LIN {X -0.027,Y -194.298,Z 687.966,A 0.000,B 0.000,C 90.000,E1 353.799} C_DIS
LIN {X 0.100,Y -197.858,Z 687.934,A 0.000,B 0.000,C 90.000,E1 348.049} C_DIS
LIN {X -0.011,Y -201.599,Z 687.911,A 0.000,B 0.000,C 90.000,E1 344.031} C_DIS
LIN {X 0.020,Y -206.301,Z 687.889,A 0.000,B 0.000,C 90.000,E1 340.007} C_DIS
LIN {X -0.035,Y -211.829,Z 687.867,A 0.000,B 0.000,C 90.000,E1 336.049} C_DIS
LIN {X 0.046,Y -218.045,Z 687.845,A 0.000,B 0.000,C 90.000,E1 332.103} C_DIS
LIN {X -0.027,Y -225.043,Z 687.824,A 0.000,B 0.000,C 90.000,E1 328.250} C_DIS
LIN {X 0.020,Y -231.035,Z 687.807,A 0.000,B 0.000,C 90.000,E1 325.182} C_DIS
LIN {X 0.033,Y -239.102,Z 687.786,A 0.000,B 0.000,C 90.000,E1 321.412} C_DIS
LIN {X 0.002,Y -248.003,Z 687.765,A 0.000,B 0.000,C 90.000,E1 317.715} C_DIS
LIN {X 0.037,Y -256.957,Z 687.747,A 0.000,B 0.000,C 90.000,E1 314.433} C_DIS
LIN {X 0.065,Y -267.947,Z 687.727,A 0.000,B 0.000,C 90.000,E1 310.862} C_DIS
LIN {X 0.020,Y -279.022,Z 687.710,A 0.000,B 0.000,C 90.000,E1 307.729} C_DIS
LIN {X -0.029,Y -292.675,Z 687.691,A 0.000,B 0.000,C 90.000,E1 304.326} C_DIS
LIN {X -0.050,Y -307.715,Z 687.672,A 0.000,B 0.000,C 90.000,E1 301.003} C_DIS
LIN {X -0.132,Y -319.136,Z 687.660,A 0.000,B 0.000,C 90.000,E1 298.743} C_DIS
LIN {X 0.084,Y -334.892,Z 687.644,A 0.000,B 0.000,C 90.000,E1 295.848} C_DIS
LIN {X 0.026,Y -351.489,Z 687.628,A 0.000,B 0.000,C 90.000,E1 293.078} C_DIS
LIN {X 0.026,Y -369.148,Z 687.613,A 0.000,B 0.000,C 90.000,E1 290.375} C_DIS
LIN {X 0.146,Y -381.918,Z 687.603,A 0.000,B 0.000,C 90.000,E1 288.598} C_DIS
LIN {X 0.106,Y -400.402,Z 687.591,A 0.000,B 0.000,C 90.000,E1 286.315} C_DIS
LIN {X -0.150,Y -412.016,Z 687.583,A 0.000,B 0.000,C 90.000,E1 284.954} C_DIS
LIN {X 0.167,Y -423.397,Z 687.575,A 0.000,B 0.000,C 90.000,E1 283.536} C_DIS
LIN {X 0.161,Y -434.292,Z 687.568,A 0.000,B 0.000,C 90.000,E1 282.187} C_DIS
LIN {X 0.099,Y -442.576,Z 687.562,A 0.000,B 0.000,C 90.000,E1 281.130} C_DIS
LIN {X -0.097,Y -460.504,Z 687.549,A 0.000,B 0.000,C 90.000,E1 278.803} C_DIS
LIN {X -0.165,Y -470.432,Z 687.542,A 0.000,B 0.000,C 90.000,E1 277.530} C_DIS
LIN {X -0.225,Y -475.757,Z 687.537,A 0.000,B 0.000,C 90.000,E1 276.777} C_DIS
LIN {X 0.239,Y -480.127,Z 687.533,A 0.000,B 0.000,C 90.000,E1 275.967} C_DIS
LIN {X 0.212,Y -483.506,Z 687.529,A 0.000,B 0.000,C 90.000,E1 275.220} C_DIS
LIN {X -0.094,Y -485.203,Z 687.526,A 0.000,B 0.000,C 90.000,E1 274.759} C_DIS
LIN {X 0.050,Y -486.474,Z 687.524,A 0.000,B 0.000,C 90.000,E1 274.245} C_DIS
LIN {X 0.241,Y -487.342,Z 687.521,A 0.000,B 0.000,C 90.000,E1 273.726} C_DIS
LIN {X -0.077,Y -487.894,Z 687.518,A 0.000,B 0.000,C 90.000,E1 273.269} C_DIS
LIN {X 0.122,Y -488.076,Z 687.515,A 0.000,B 0.000,C 90.000,E1 272.751} C_DIS
LIN {X -0.186,Y -487.966,Z 687.513,A 0.000,B 0.000,C 90.000,E1 272.293} C_DIS
LIN {X 0.013,Y -487.497,Z 687.510,A 0.000,B 0.000,C 90.000,E1 271.776} C_DIS
LIN {X 0.193,Y -486.720,Z 687.507,A 0.000,B 0.000,C 90.000,E1 271.260} C_DIS
LIN {X -0.115,Y -485.520,Z 687.504,A 0.000,B 0.000,C 90.000,E1 270.802} C_DIS
LIN {X 0.061,Y -483.850,Z 687.502,A 0.000,B 0.000,C 90.000,E1 270.286} C_DIS
LIN {X 0.228,Y -481.575,Z 687.499,A 0.000,B 0.000,C 90.000,E1 269.771} C_DIS
LIN {X 0.063,Y -480.227,Z 687.497,A 0.000,B 0.000,C 90.000,E1 269.542} C_DIS
LIN {X 0.206,Y -476.929,Z 687.495,A 0.000,B 0.000,C 90.000,E1 269.026} C_DIS
LIN {X -0.145,Y -472.762,Z 687.492,A 0.000,B 0.000,C 90.000,E1 268.568} C_DIS
LIN {X 0.005,Y -467.541,Z 687.489,A 0.000,B 0.000,C 90.000,E1 268.051} C_DIS
LIN {X -0.015,Y -461.447,Z 687.487,A 0.000,B 0.000,C 90.000,E1 267.593} C_DIS
LIN {X 0.115,Y -458.008,Z 687.485,A 0.000,B 0.000,C 90.000,E1 267.364} C_DIS
LIN {X 0.027,Y -451.055,Z 687.483,A 0.000,B 0.000,C 90.000,E1 267.020} C_DIS
LIN {X 0.028,Y -443.900,Z 687.482,A 0.000,B 0.000,C 90.000,E1 266.731} C_DIS
LIN {X 0.017,Y -436.381,Z 687.481,A 0.000,B 0.000,C 90.000,E1 266.502} C_DIS
LIN {X 0.206,Y -432.252,Z 687.480,A 0.000,B 0.000,C 90.000,E1 266.388} C_DIS
LIN {X 0.052,Y -421.992,Z 687.479,A 0.000,B 0.000,C 90.000,E1 266.274} C_DIS
LIN {X -0.200,Y -415.695,Z 687.479,A 0.000,B 0.000,C 90.000,E1 266.274} C_DIS
LIN {X 0.071,Y -180.932,Z 687.479,A 0.000,B 0.000,C 90.000,E1 266.216} C_DIS
LIN {X -0.053,Y -180.770,Z 687.471,A 0.000,B 0.000,C 90.000,E1 264.723} C_DIS
LIN {X -0.015,Y -178.987,Z 687.444,A 0.000,B 0.000,C 90.000,E1 259.982} C_DIS
LIN {X -0.004,Y -177.967,Z 687.435,A 0.000,B 0.000,C 90.000,E1 258.285} C_DIS
LIN {X 0.015,Y -175.610,Z 687.411,A 0.000,B 0.000,C 90.000,E1 254.031} C_DIS
LIN {X 0.027,Y -172.332,Z 687.388,A 0.000,B 0.000,C 90.000,E1 249.752} C_DIS
LIN {X 0.006,Y -171.808,Z 687.383,A 0.000,B 0.000,C 90.000,E1 248.901} C_DIS
LIN {X 0.013,Y -170.270,Z 687.373,A 0.000,B 0.000,C 90.000,E1 247.177} C_DIS
LIN {X -0.051,Y -166.812,Z 687.349,A 0.000,B 0.000,C 90.000,E1 242.871} C_DIS
LIN {X 0.007,Y -162.794,Z 687.325,A 0.000,B 0.000,C 90.000,E1 238.486} C_DIS
LIN {X 0.067,Y -161.481,Z 687.315,A 0.000,B 0.000,C 90.000,E1 236.707} C_DIS
LIN {X -0.017,Y -157.477,Z 687.291,A 0.000,B 0.000,C 90.000,E1 232.316} C_DIS
LIN {X 0.040,Y -155.493,Z 687.276,A 0.000,B 0.000,C 90.000,E1 229.622} C_DIS
LIN {X -0.028,Y -151.799,Z 687.251,A 0.000,B 0.000,C 90.000,E1 225.162} C_DIS
LIN {X -0.015,Y -150.008,Z 687.236,A 0.000,B 0.000,C 90.000,E1 222.447} C_DIS
LIN {X 0.017,Y -146.834,Z 687.211,A 0.000,B 0.000,C 90.000,E1 217.890} C_DIS
LIN {X 0.003,Y -145.416,Z 687.195,A 0.000,B 0.000,C 90.000,E1 215.152} C_DIS
LIN {X 0.038,Y -142.844,Z 687.170,A 0.000,B 0.000,C 90.000,E1 210.541} C_DIS
LIN {X -0.032,Y -141.458,Z 687.149,A 0.000,B 0.000,C 90.000,E1 206.873} C_DIS
LIN {X 0.008,Y -139.374,Z 687.113,A 0.000,B 0.000,C 90.000,E1 200.355} C_DIS
LIN {X -0.051,Y -138.825,Z 687.098,A 0.000,B 0.000,C 90.000,E1 197.583} C_DIS
LIN {X 0.038,Y -138.353,Z 687.056,A 0.000,B 0.000,C 90.000,E1 190.074} C_DIS
LIN {X 0.012,Y -139.531,Z 687.004,A 0.000,B 0.000,C 90.000,E1 180.745} C_DIS
LIN {X -0.036,Y -141.212,Z 686.973,A 0.000,B 0.000,C 90.000,E1 175.179} C_DIS
LIN {X 0.065,Y -142.585,Z 686.958,A 0.000,B 0.000,C 90.000,E1 172.356} C_DIS
LIN {X 0.019,Y -144.883,Z 686.932,A 0.000,B 0.000,C 90.000,E1 167.757} C_DIS
LIN {X -0.028,Y -147.510,Z 686.912,A 0.000,B 0.000,C 90.000,E1 164.102} C_DIS
LIN {X 0.047,Y -150.103,Z 686.891,A 0.000,B 0.000,C 90.000,E1 160.423} C_DIS
LIN {X 0.059,Y -153.461,Z 686.871,A 0.000,B 0.000,C 90.000,E1 156.794} C_DIS
LIN {X -0.089,Y -157.823,Z 686.846,A 0.000,B 0.000,C 90.000,E1 152.359} C_DIS
LIN {X -0.057,Y -162.107,Z 686.826,A 0.000,B 0.000,C 90.000,E1 148.791} C_DIS
LIN {X -0.033,Y -166.308,Z 686.807,A 0.000,B 0.000,C 90.000,E1 145.261} C_DIS
LIN {X 0.069,Y -171.325,Z 686.788,A 0.000,B 0.000,C 90.000,E1 141.743} C_DIS
LIN {X -0.003,Y -176.225,Z 686.768,A 0.000,B 0.000,C 90.000,E1 138.324} C_DIS
LIN {X -0.009,Y -180.504,Z 686.754,A 0.000,B 0.000,C 90.000,E1 135.769} C_DIS
LIN {X 0.097,Y -185.907,Z 686.736,A 0.000,B 0.000,C 90.000,E1 132.366} C_DIS
LIN {X 0.078,Y -191.207,Z 686.719,A 0.000,B 0.000,C 90.000,E1 129.483} C_DIS
LIN {X 0.075,Y -289.233,Z 686.719,A 0.000,B 0.000,C 90.000,E1 129.483} C_DIS
LIN {X 0.007,Y -295.104,Z 686.718,A 0.000,B 0.000,C 90.000,E1 129.277} C_DIS
LIN {X -0.016,Y -297.647,Z 686.717,A 0.000,B 0.000,C 90.000,E1 129.072} C_DIS
LIN {X -0.033,Y -301.459,Z 686.714,A 0.000,B 0.000,C 90.000,E1 128.588} C_DIS
LIN {X -0.038,Y -303.267,Z 686.713,A 0.000,B 0.000,C 90.000,E1 128.257} C_DIS
LIN {X -0.094,Y -304.679,Z 686.711,A 0.000,B 0.000,C 90.000,E1 127.935} C_DIS
LIN {X 0.123,Y -306.687,Z 686.707,A 0.000,B 0.000,C 90.000,E1 127.237} C_DIS
LIN {X 0.057,Y -316.400,Z 686.689,A 0.000,B 0.000,C 90.000,E1 123.992} C_DIS
LIN {X -0.038,Y -326.433,Z 686.673,A 0.000,B 0.000,C 90.000,E1 121.131} C_DIS
LIN {X 0.089,Y -337.794,Z 686.657,A 0.000,B 0.000,C 90.000,E1 118.281} C_DIS
LIN {X -0.088,Y -350.581,Z 686.642,A 0.000,B 0.000,C 90.000,E1 115.540} C_DIS
LIN {X -0.118,Y -363.240,Z 686.628,A 0.000,B 0.000,C 90.000,E1 113.131} C_DIS
LIN {X 0.082,Y -377.206,Z 686.615,A 0.000,B 0.000,C 90.000,E1 110.737} C_DIS
LIN {X 0.160,Y -392.584,Z 686.602,A 0.000,B 0.000,C 90.000,E1 108.417} C_DIS
LIN {X -0.133,Y -409.482,Z 686.590,A 0.000,B 0.000,C 90.000,E1 106.205} C_DIS
LIN {X -0.128,Y -428.026,Z 686.578,A 0.000,B 0.000,C 90.000,E1 104.008} C_DIS
LIN {X 0.121,Y -447.934,Z 686.566,A 0.000,B 0.000,C 90.000,E1 101.883} C_DIS
LIN {X 0.120,Y -468.437,Z 686.555,A 0.000,B 0.000,C 90.000,E1 99.962} C_DIS
LIN {X 0.167,Y -470.660,Z 686.554,A 0.000,B 0.000,C 90.000,E1 99.726} C_DIS
LIN {X -0.052,Y -472.481,Z 686.553,A 0.000,B 0.000,C 90.000,E1 99.500} C_DIS
LIN {X -0.192,Y -473.850,Z 686.551,A 0.000,B 0.000,C 90.000,E1 99.265} C_DIS
LIN {X -0.079,Y -475.584,Z 686.549,A 0.000,B 0.000,C 90.000,E1 98.746} C_DIS
LIN {X 0.115,Y -476.240,Z 686.546,A 0.000,B 0.000,C 90.000,E1 98.219} C_DIS
LIN {X -0.224,Y -475.928,Z 686.543,A 0.000,B 0.000,C 90.000,E1 97.757} C_DIS
LIN {X -0.085,Y -474.605,Z 686.540,A 0.000,B 0.000,C 90.000,E1 97.239} C_DIS
LIN {X 0.247,Y -473.499,Z 686.539,A 0.000,B 0.000,C 90.000,E1 96.947} C_DIS
LIN {X 0.053,Y -472.021,Z 686.537,A 0.000,B 0.000,C 90.000,E1 96.720} C_DIS
LIN {X 0.219,Y -453.746,Z 686.522,A 0.000,B 0.000,C 90.000,E1 93.898} C_DIS
LIN {X 0.187,Y -437.541,Z 686.506,A 0.000,B 0.000,C 90.000,E1 91.031} C_DIS
LIN {X 0.114,Y -430.195,Z 686.498,A 0.000,B 0.000,C 90.000,E1 89.714} C_DIS
LIN {X 0.071,Y -420.954,Z 686.490,A 0.000,B 0.000,C 90.000,E1 88.108} C_DIS
LIN {X 0.059,Y -408.465,Z 686.477,A 0.000,B 0.000,C 90.000,E1 85.927} C_DIS
LIN {X 0.177,Y -395.953,Z 686.465,A 0.000,B 0.000,C 90.000,E1 83.685} C_DIS
LIN {X 0.115,Y -382.283,Z 686.451,A 0.000,B 0.000,C 90.000,E1 81.141} C_DIS
LIN {X 0.186,Y -370.570,Z 686.438,A 0.000,B 0.000,C 90.000,E1 78.814} C_DIS
LIN {X 0.043,Y -356.463,Z 686.422,A 0.000,B 0.000,C 90.000,E1 75.880} C_DIS
LIN {X -0.177,Y -345.659,Z 686.408,A 0.000,B 0.000,C 90.000,E1 73.504} C_DIS
LIN {X -0.138,Y -333.972,Z 686.393,A 0.000,B 0.000,C 90.000,E1 70.732} C_DIS
LIN {X 0.076,Y -319.540,Z 686.372,A 0.000,B 0.000,C 90.000,E1 66.922} C_DIS
LIN {X 0.089,Y -307.949,Z 686.352,A 0.000,B 0.000,C 90.000,E1 63.384} C_DIS
LIN {X -0.001,Y -298.482,Z 686.334,A 0.000,B 0.000,C 90.000,E1 60.127} C_DIS
LIN {X 0.061,Y -289.725,Z 686.316,A 0.000,B 0.000,C 90.000,E1 56.786} C_DIS
LIN {X -0.091,Y -283.065,Z 686.301,A 0.000,B 0.000,C 90.000,E1 54.116} C_DIS
LIN {X -0.074,Y -278.087,Z 686.289,A 0.000,B 0.000,C 90.000,E1 52.065} C_DIS
LIN {X -0.031,Y -272.884,Z 686.278,A 0.000,B 0.000,C 90.000,E1 49.989} C_DIS
LIN {X -0.112,Y -267.376,Z 686.266,A 0.000,B 0.000,C 90.000,E1 47.919} C_DIS
LIN {X -0.112,Y -261.484,Z 686.254,A 0.000,B 0.000,C 90.000,E1 45.810} C_DIS
LIN {X 0.132,Y -255.455,Z 686.242,A 0.000,B 0.000,C 90.000,E1 43.623} C_DIS
LIN {X -0.093,Y -249.280,Z 686.231,A 0.000,B 0.000,C 90.000,E1 41.515} C_DIS
LIN {X 0.129,Y -242.951,Z 686.218,A 0.000,B 0.000,C 90.000,E1 39.277} C_DIS
LIN {X 0.026,Y -232.833,Z 686.198,A 0.000,B 0.000,C 90.000,E1 35.598} C_DIS
LIN {X -0.033,Y -225.322,Z 686.181,A 0.000,B 0.000,C 90.000,E1 32.594} C_DIS
LIN {X -0.067,Y -218.723,Z 686.164,A 0.000,B 0.000,C 90.000,E1 29.539} C_DIS
LIN {X 0.010,Y -212.830,Z 686.147,A 0.000,B 0.000,C 90.000,E1 26.411} C_DIS
LIN {X 0.035,Y -207.796,Z 686.129,A 0.000,B 0.000,C 90.000,E1 23.259} C_DIS
LIN {X 0.076,Y -202.633,Z 686.107,A 0.000,B 0.000,C 90.000,E1 19.268} C_DIS
LIN {X 0.080,Y -198.620,Z 686.085,A 0.000,B 0.000,C 90.000,E1 15.245} C_DIS
LIN {X 0.109,Y -195.196,Z 686.058,A 0.000,B 0.000,C 90.000,E1 10.366} C_DIS
LIN {X -0.002,Y -192.827,Z 686.017,A 0.000,B 0.000,C 90.000,E1 3.037} C_DIS
LIN {X -0.022,Y -194.394,Z 685.966,A 0.000,B 0.000,C 90.000,E1 353.799} C_DIS
LIN {X 0.109,Y -197.929,Z 685.934,A 0.000,B 0.000,C 90.000,E1 348.049} C_DIS
LIN {X 0.001,Y -201.671,Z 685.911,A 0.000,B 0.000,C 90.000,E1 344.031} C_DIS
LIN {X 0.034,Y -206.368,Z 685.889,A 0.000,B 0.000,C 90.000,E1 340.007} C_DIS
LIN {X -0.019,Y -211.878,Z 685.867,A 0.000,B 0.000,C 90.000,E1 336.049} C_DIS
LIN {X 0.064,Y -218.099,Z 685.845,A 0.000,B 0.000,C 90.000,E1 332.103} C_DIS
LIN {X -0.007,Y -225.100,Z 685.824,A 0.000,B 0.000,C 90.000,E1 328.250} C_DIS
LIN {X 0.042,Y -231.081,Z 685.807,A 0.000,B 0.000,C 90.000,E1 325.182} C_DIS
LIN {X 0.057,Y -239.126,Z 685.786,A 0.000,B 0.000,C 90.000,E1 321.412} C_DIS
LIN {X 0.029,Y -248.003,Z 685.765,A 0.000,B 0.000,C 90.000,E1 317.715} C_DIS
LIN {X -0.096,Y -258.017,Z 685.745,A 0.000,B 0.000,C 90.000,E1 314.109} C_DIS
LIN {X -0.044,Y -269.115,Z 685.725,A 0.000,B 0.000,C 90.000,E1 310.539} C_DIS
LIN {X -0.013,Y -280.316,Z 685.708,A 0.000,B 0.000,C 90.000,E1 307.397} C_DIS
LIN {X -0.011,Y -294.084,Z 685.689,A 0.000,B 0.000,C 90.000,E1 303.992} C_DIS
LIN {X 0.019,Y -309.250,Z 685.670,A 0.000,B 0.000,C 90.000,E1 300.669} C_DIS
LIN {X -0.091,Y -326.003,Z 685.652,A 0.000,B 0.000,C 90.000,E1 297.462} C_DIS
LIN {X -0.121,Y -342.118,Z 685.637,A 0.000,B 0.000,C 90.000,E1 294.643} C_DIS
LIN {X -0.018,Y -363.058,Z 685.618,A 0.000,B 0.000,C 90.000,E1 291.280} C_DIS
LIN {X -0.018,Y -375.260,Z 685.608,A 0.000,B 0.000,C 90.000,E1 289.504} C_DIS
LIN {X -0.083,Y -395.523,Z 685.594,A 0.000,B 0.000,C 90.000,E1 286.913} C_DIS
LIN {X 0.174,Y -409.571,Z 685.585,A 0.000,B 0.000,C 90.000,E1 285.190} C_DIS
LIN {X -0.216,Y -423.240,Z 685.575,A 0.000,B 0.000,C 90.000,E1 283.592} C_DIS
LIN {X -0.237,Y -434.130,Z 685.568,A 0.000,B 0.000,C 90.000,E1 282.243} C_DIS
LIN {X 0.123,Y -442.396,Z 685.562,A 0.000,B 0.000,C 90.000,E1 281.130} C_DIS
LIN {X 0.202,Y -462.319,Z 685.547,A 0.000,B 0.000,C 90.000,E1 278.511} C_DIS
LIN {X -0.147,Y -470.230,Z 685.542,A 0.000,B 0.000,C 90.000,E1 277.530} C_DIS
LIN {X -0.208,Y -475.560,Z 685.538,A 0.000,B 0.000,C 90.000,E1 276.777} C_DIS
LIN {X -0.082,Y -478.576,Z 685.535,A 0.000,B 0.000,C 90.000,E1 276.258} C_DIS
LIN {X -0.119,Y -482.284,Z 685.531,A 0.000,B 0.000,C 90.000,E1 275.511} C_DIS
LIN {X -0.082,Y -484.984,Z 685.526,A 0.000,B 0.000,C 90.000,E1 274.759} C_DIS
LIN {X 0.060,Y -486.297,Z 685.524,A 0.000,B 0.000,C 90.000,E1 274.245} C_DIS
LIN {X -0.235,Y -487.161,Z 685.521,A 0.000,B 0.000,C 90.000,E1 273.784} C_DIS
LIN {X -0.070,Y -487.709,Z 685.518,A 0.000,B 0.000,C 90.000,E1 273.269} C_DIS
LIN {X 0.129,Y -487.921,Z 685.515,A 0.000,B 0.000,C 90.000,E1 272.751} C_DIS
LIN {X -0.180,Y -487.837,Z 685.513,A 0.000,B 0.000,C 90.000,E1 272.293} C_DIS
LIN {X 0.018,Y -487.439,Z 685.510,A 0.000,B 0.000,C 90.000,E1 271.776} C_DIS
LIN {X 0.198,Y -486.637,Z 685.507,A 0.000,B 0.000,C 90.000,E1 271.260} C_DIS
LIN {X -0.110,Y -485.469,Z 685.504,A 0.000,B 0.000,C 90.000,E1 270.802} C_DIS
LIN {X 0.065,Y -483.831,Z 685.502,A 0.000,B 0.000,C 90.000,E1 270.286} C_DIS
LIN {X 0.231,Y -481.597,Z 685.499,A 0.000,B 0.000,C 90.000,E1 269.771} C_DIS
LIN {X -0.097,Y -478.673,Z 685.496,A 0.000,B 0.000,C 90.000,E1 269.312} C_DIS
LIN {X 0.208,Y -476.971,Z 685.495,A 0.000,B 0.000,C 90.000,E1 269.026} C_DIS
LIN {X -0.142,Y -472.795,Z 685.492,A 0.000,B 0.000,C 90.000,E1 268.568} C_DIS
LIN {X 0.013,Y -467.555,Z 685.489,A 0.000,B 0.000,C 90.000,E1 268.051} C_DIS
LIN {X -0.015,Y -461.461,Z 685.487,A 0.000,B 0.000,C 90.000,E1 267.593} C_DIS
LIN {X 0.051,Y -454.772,Z 685.484,A 0.000,B 0.000,C 90.000,E1 267.192} C_DIS
LIN {X -0.226,Y -447.733,Z 685.483,A 0.000,B 0.000,C 90.000,E1 266.906} C_DIS
LIN {X 0.004,Y -440.474,Z 685.481,A 0.000,B 0.000,C 90.000,E1 266.617} C_DIS
LIN {X 0.194,Y -432.352,Z 685.480,A 0.000,B 0.000,C 90.000,E1 266.388} C_DIS
LIN {X 0.061,Y -422.993,Z 685.479,A 0.000,B 0.000,C 90.000,E1 266.274} C_DIS
LIN {X 0.153,Y -415.264,Z 685.479,A 0.000,B 0.000,C 90.000,E1 266.216} C_DIS
LIN {X 0.043,Y -180.931,Z 685.479,A 0.000,B 0.000,C 90.000,E1 266.216} C_DIS
LIN {X -0.061,Y -180.769,Z 685.471,A 0.000,B 0.000,C 90.000,E1 264.723} C_DIS
LIN {X -0.024,Y -178.986,Z 685.444,A 0.000,B 0.000,C 90.000,E1 259.982} C_DIS
LIN {X -0.012,Y -177.965,Z 685.435,A 0.000,B 0.000,C 90.000,E1 258.285} C_DIS
LIN {X 0.007,Y -175.608,Z 685.411,A 0.000,B 0.000,C 90.000,E1 254.031} C_DIS
LIN {X 0.020,Y -172.330,Z 685.388,A 0.000,B 0.000,C 90.000,E1 249.752} C_DIS
LIN {X -0.001,Y -171.807,Z 685.383,A 0.000,B 0.000,C 90.000,E1 248.901} C_DIS
LIN {X 0.006,Y -170.268,Z 685.373,A 0.000,B 0.000,C 90.000,E1 247.177} C_DIS
LIN {X -0.058,Y -166.810,Z 685.349,A 0.000,B 0.000,C 90.000,E1 242.871} C_DIS
LIN {X 0.000,Y -162.792,Z 685.325,A 0.000,B 0.000,C 90.000,E1 238.486} C_DIS
LIN {X 0.060,Y -161.480,Z 685.315,A 0.000,B 0.000,C 90.000,E1 236.707} C_DIS
LIN {X -0.024,Y -157.475,Z 685.291,A 0.000,B 0.000,C 90.000,E1 232.316} C_DIS
LIN {X 0.033,Y -155.490,Z 685.276,A 0.000,B 0.000,C 90.000,E1 229.622} C_DIS
LIN {X -0.034,Y -151.797,Z 685.251,A 0.000,B 0.000,C 90.000,E1 225.162} C_DIS
LIN {X -0.021,Y -150.006,Z 685.236,A 0.000,B 0.000,C 90.000,E1 222.447} C_DIS
LIN {X 0.010,Y -146.833,Z 685.211,A 0.000,B 0.000,C 90.000,E1 217.890} C_DIS
LIN {X -0.004,Y -145.413,Z 685.195,A 0.000,B 0.000,C 90.000,E1 215.152} C_DIS
LIN {X 0.032,Y -142.843,Z 685.170,A 0.000,B 0.000,C 90.000,E1 210.541} C_DIS
LIN {X -0.039,Y -141.457,Z 685.149,A 0.000,B 0.000,C 90.000,E1 206.873} C_DIS
LIN {X 0.001,Y -139.373,Z 685.113,A 0.000,B 0.000,C 90.000,E1 200.355} C_DIS
LIN {X -0.057,Y -138.824,Z 685.098,A 0.000,B 0.000,C 90.000,E1 197.583} C_DIS
LIN {X 0.032,Y -138.353,Z 685.056,A 0.000,B 0.000,C 90.000,E1 190.074} C_DIS
LIN {X 0.005,Y -139.532,Z 685.004,A 0.000,B 0.000,C 90.000,E1 180.745} C_DIS
LIN {X -0.042,Y -141.212,Z 684.973,A 0.000,B 0.000,C 90.000,E1 175.179} C_DIS
LIN {X 0.058,Y -142.586,Z 684.958,A 0.000,B 0.000,C 90.000,E1 172.356} C_DIS
LIN {X 0.012,Y -144.885,Z 684.932,A 0.000,B 0.000,C 90.000,E1 167.757} C_DIS
LIN {X -0.035,Y -147.512,Z 684.912,A 0.000,B 0.000,C 90.000,E1 164.102} C_DIS
LIN {X 0.040,Y -150.106,Z 684.891,A 0.000,B 0.000,C 90.000,E1 160.423} C_DIS
LIN {X 0.053,Y -153.462,Z 684.871,A 0.000,B 0.000,C 90.000,E1 156.794} C_DIS
LIN {X -0.096,Y -157.826,Z 684.846,A 0.000,B 0.000,C 90.000,E1 152.359} C_DIS
LIN {X 0.074,Y -162.110,Z 684.826,A 0.000,B 0.000,C 90.000,E1 148.742} C_DIS
LIN {X -0.040,Y -166.311,Z 684.807,A 0.000,B 0.000,C 90.000,E1 145.261} C_DIS
LIN {X 0.061,Y -171.329,Z 684.788,A 0.000,B 0.000,C 90.000,E1 141.743} C_DIS
LIN {X -0.010,Y -176.229,Z 684.768,A 0.000,B 0.000,C 90.000,E1 138.324} C_DIS
LIN {X 0.109,Y -180.509,Z 684.754,A 0.000,B 0.000,C 90.000,E1 135.729} C_DIS
LIN {X 0.089,Y -185.911,Z 684.736,A 0.000,B 0.000,C 90.000,E1 132.366} C_DIS
LIN {X 0.006,Y -191.183,Z 684.720,A 0.000,B 0.000,C 90.000,E1 129.519} C_DIS
LIN {X -0.034,Y -288.963,Z 684.720,A 0.000,B 0.000,C 90.000,E1 129.519} C_DIS
LIN {X 0.020,Y -290.728,Z 684.719,A 0.000,B 0.000,C 90.000,E1 129.483} C_DIS
LIN {X -0.005,Y -295.281,Z 684.718,A 0.000,B 0.000,C 90.000,E1 129.277} C_DIS
LIN {X -0.028,Y -297.754,Z 684.717,A 0.000,B 0.000,C 90.000,E1 129.072} C_DIS
LIN {X 0.129,Y -301.574,Z 684.714,A 0.000,B 0.000,C 90.000,E1 128.543} C_DIS
LIN {X -0.112,Y -303.342,Z 684.712,A 0.000,B 0.000,C 90.000,E1 128.257} C_DIS
LIN {X 0.073,Y -304.726,Z 684.711,A 0.000,B 0.000,C 90.000,E1 127.890} C_DIS
LIN {X 0.034,Y -308.532,Z 684.703,A 0.000,B 0.000,C 90.000,E1 126.583} C_DIS
LIN {X -0.153,Y -318.544,Z 684.685,A 0.000,B 0.000,C 90.000,E1 123.372} C_DIS
LIN {X 0.086,Y -328.870,Z 684.669,A 0.000,B 0.000,C 90.000,E1 120.463} C_DIS
LIN {X 0.125,Y -340.546,Z 684.654,A 0.000,B 0.000,C 90.000,E1 117.641} C_DIS
LIN {X 0.032,Y -353.672,Z 684.638,A 0.000,B 0.000,C 90.000,E1 114.899} C_DIS
LIN {X -0.066,Y -366.655,Z 684.625,A 0.000,B 0.000,C 90.000,E1 112.514} C_DIS
LIN {X -0.131,Y -380.973,Z 684.612,A 0.000,B 0.000,C 90.000,E1 110.174} C_DIS
LIN {X -0.101,Y -396.727,Z 684.599,A 0.000,B 0.000,C 90.000,E1 107.873} C_DIS
LIN {X 0.093,Y -414.034,Z 684.587,A 0.000,B 0.000,C 90.000,E1 105.607} C_DIS
LIN {X 0.226,Y -433.008,Z 684.575,A 0.000,B 0.000,C 90.000,E1 103.411} C_DIS
LIN {X -0.248,Y -453.095,Z 684.563,A 0.000,B 0.000,C 90.000,E1 101.422} C_DIS
LIN {X 0.035,Y -468.525,Z 684.555,A 0.000,B 0.000,C 90.000,E1 99.962} C_DIS
LIN {X 0.081,Y -470.740,Z 684.554,A 0.000,B 0.000,C 90.000,E1 99.726} C_DIS
LIN {X -0.142,Y -472.558,Z 684.553,A 0.000,B 0.000,C 90.000,E1 99.500} C_DIS
LIN {X 0.182,Y -473.925,Z 684.551,A 0.000,B 0.000,C 90.000,E1 99.208} C_DIS
LIN {X -0.173,Y -475.650,Z 684.548,A 0.000,B 0.000,C 90.000,E1 98.746} C_DIS
LIN {X 0.021,Y -476.299,Z 684.546,A 0.000,B 0.000,C 90.000,E1 98.219} C_DIS
LIN {X 0.155,Y -475.982,Z 684.543,A 0.000,B 0.000,C 90.000,E1 97.701} C_DIS
LIN {X -0.177,Y -474.652,Z 684.540,A 0.000,B 0.000,C 90.000,E1 97.239} C_DIS
LIN {X 0.155,Y -473.541,Z 684.539,A 0.000,B 0.000,C 90.000,E1 96.947} C_DIS
LIN {X -0.185,Y -470.334,Z 684.536,A 0.000,B 0.000,C 90.000,E1 96.486} C_DIS
LIN {X 0.132,Y -453.752,Z 684.522,A 0.000,B 0.000,C 90.000,E1 93.898} C_DIS
LIN {X 0.103,Y -437.573,Z 684.506,A 0.000,B 0.000,C 90.000,E1 91.031} C_DIS
LIN {X 0.032,Y -430.237,Z 684.498,A 0.000,B 0.000,C 90.000,E1 89.714} C_DIS
LIN {X -0.009,Y -420.997,Z 684.490,A 0.000,B 0.000,C 90.000,E1 88.108} C_DIS
LIN {X -0.018,Y -408.503,Z 684.477,A 0.000,B 0.000,C 90.000,E1 85.927} C_DIS
LIN {X 0.176,Y -394.472,Z 684.463,A 0.000,B 0.000,C 90.000,E1 83.394} C_DIS
LIN {X 0.107,Y -379.419,Z 684.448,A 0.000,B 0.000,C 90.000,E1 80.557} C_DIS
LIN {X 0.100,Y -366.375,Z 684.433,A 0.000,B 0.000,C 90.000,E1 77.937} C_DIS
LIN {X -0.047,Y -351.160,Z 684.415,A 0.000,B 0.000,C 90.000,E1 74.685} C_DIS
LIN {X -0.057,Y -337.973,Z 684.398,A 0.000,B 0.000,C 90.000,E1 71.638} C_DIS
LIN {X -0.077,Y -324.350,Z 684.379,A 0.000,B 0.000,C 90.000,E1 68.209} C_DIS
LIN {X -0.152,Y -314.276,Z 684.363,A 0.000,B 0.000,C 90.000,E1 65.357} C_DIS
LIN {X 0.012,Y -302.398,Z 684.341,A 0.000,B 0.000,C 90.000,E1 61.435} C_DIS
LIN {X 0.051,Y -293.396,Z 684.323,A 0.000,B 0.000,C 90.000,E1 58.122} C_DIS
LIN {X 0.023,Y -284.997,Z 684.304,A 0.000,B 0.000,C 90.000,E1 54.769} C_DIS
LIN {X 0.073,Y -280.025,Z 684.293,A 0.000,B 0.000,C 90.000,E1 52.718} C_DIS
LIN {X -0.025,Y -274.898,Z 684.281,A 0.000,B 0.000,C 90.000,E1 50.678} C_DIS
LIN {X -0.073,Y -269.532,Z 684.270,A 0.000,B 0.000,C 90.000,E1 48.609} C_DIS
LIN {X -0.033,Y -263.753,Z 684.258,A 0.000,B 0.000,C 90.000,E1 46.500} C_DIS
LIN {X 0.076,Y -257.707,Z 684.247,A 0.000,B 0.000,C 90.000,E1 44.352} C_DIS
LIN {X 0.065,Y -251.568,Z 684.235,A 0.000,B 0.000,C 90.000,E1 42.204} C_DIS
LIN {X 0.141,Y -245.296,Z 684.222,A 0.000,B 0.000,C 90.000,E1 40.011} C_DIS
LIN {X -0.082,Y -234.986,Z 684.202,A 0.000,B 0.000,C 90.000,E1 36.377} C_DIS
LIN {X -0.079,Y -227.320,Z 684.185,A 0.000,B 0.000,C 90.000,E1 33.372} C_DIS
LIN {X -0.135,Y -220.477,Z 684.168,A 0.000,B 0.000,C 90.000,E1 30.335} C_DIS
LIN {X -0.006,Y -214.406,Z 684.151,A 0.000,B 0.000,C 90.000,E1 27.206} C_DIS
LIN {X -0.035,Y -209.129,Z 684.134,A 0.000,B 0.000,C 90.000,E1 24.079} C_DIS
LIN {X -0.066,Y -203.753,Z 684.112,A 0.000,B 0.000,C 90.000,E1 20.120} C_DIS
LIN {X 0.036,Y -199.512,Z 684.089,A 0.000,B 0.000,C 90.000,E1 16.079} C_DIS
LIN {X -0.048,Y -195.832,Z 684.062,A 0.000,B 0.000,C 90.000,E1 11.243} C_DIS
LIN {X -0.026,Y -193.177,Z 684.026,A 0.000,B 0.000,C 90.000,E1 4.702} C_DIS
LIN {X -0.017,Y -194.487,Z 683.966,A 0.000,B 0.000,C 90.000,E1 353.799} C_DIS
LIN {X -0.076,Y -198.006,Z 683.934,A 0.000,B 0.000,C 90.000,E1 348.105} C_DIS
LIN {X 0.011,Y -201.743,Z 683.911,A 0.000,B 0.000,C 90.000,E1 344.031} C_DIS
LIN {X 0.047,Y -206.434,Z 683.889,A 0.000,B 0.000,C 90.000,E1 340.007} C_DIS
LIN {X -0.003,Y -211.932,Z 683.867,A 0.000,B 0.000,C 90.000,E1 336.049} C_DIS
LIN {X 0.083,Y -218.158,Z 683.845,A 0.000,B 0.000,C 90.000,E1 332.103} C_DIS
LIN {X 0.014,Y -225.152,Z 683.824,A 0.000,B 0.000,C 90.000,E1 328.250} C_DIS
LIN {X 0.065,Y -231.113,Z 683.807,A 0.000,B 0.000,C 90.000,E1 325.182} C_DIS
LIN {X -0.105,Y -239.152,Z 683.786,A 0.000,B 0.000,C 90.000,E1 321.457} C_DIS
LIN {X 0.055,Y -248.026,Z 683.765,A 0.000,B 0.000,C 90.000,E1 317.715} C_DIS
LIN {X -0.069,Y -258.038,Z 683.745,A 0.000,B 0.000,C 90.000,E1 314.109} C_DIS
LIN {X -0.016,Y -269.103,Z 683.725,A 0.000,B 0.000,C 90.000,E1 310.539} C_DIS
LIN {X 0.017,Y -280.297,Z 683.708,A 0.000,B 0.000,C 90.000,E1 307.397} C_DIS
LIN {X 0.020,Y -294.089,Z 683.689,A 0.000,B 0.000,C 90.000,E1 303.992} C_DIS
LIN {X 0.051,Y -309.221,Z 683.670,A 0.000,B 0.000,C 90.000,E1 300.669} C_DIS
LIN {X -0.059,Y -325.973,Z 683.653,A 0.000,B 0.000,C 90.000,E1 297.462} C_DIS
LIN {X -0.073,Y -340.227,Z 683.639,A 0.000,B 0.000,C 90.000,E1 294.951} C_DIS
LIN {X 0.155,Y -355.114,Z 683.625,A 0.000,B 0.000,C 90.000,E1 292.461} C_DIS
LIN {X 0.013,Y -375.131,Z 683.608,A 0.000,B 0.000,C 90.000,E1 289.504} C_DIS
LIN {X -0.205,Y -393.039,Z 683.596,A 0.000,B 0.000,C 90.000,E1 287.221} C_DIS
LIN {X 0.114,Y -407.100,Z 683.586,A 0.000,B 0.000,C 90.000,E1 285.481} C_DIS
LIN {X 0.085,Y -420.827,Z 683.577,A 0.000,B 0.000,C 90.000,E1 283.828} C_DIS
LIN {X 0.029,Y -431.821,Z 683.569,A 0.000,B 0.000,C 90.000,E1 282.479} C_DIS
LIN {X -0.065,Y -440.240,Z 683.563,A 0.000,B 0.000,C 90.000,E1 281.422} C_DIS
LIN {X 0.136,Y -454.044,Z 683.553,A 0.000,B 0.000,C 90.000,E1 279.557} C_DIS
LIN {X -0.196,Y -466.148,Z 683.545,A 0.000,B 0.000,C 90.000,E1 278.049} C_DIS
LIN {X 0.174,Y -471.877,Z 683.540,A 0.000,B 0.000,C 90.000,E1 277.239} C_DIS
LIN {X -0.193,Y -475.309,Z 683.538,A 0.000,B 0.000,C 90.000,E1 276.777} C_DIS
LIN {X -0.069,Y -478.368,Z 683.535,A 0.000,B 0.000,C 90.000,E1 276.258} C_DIS
LIN {X 0.076,Y -480.952,Z 683.532,A 0.000,B 0.000,C 90.000,E1 275.739} C_DIS
LIN {X 0.238,Y -483.087,Z 683.529,A 0.000,B 0.000,C 90.000,E1 275.220} C_DIS
LIN {X -0.071,Y -484.820,Z 683.526,A 0.000,B 0.000,C 90.000,E1 274.759} C_DIS
LIN {X 0.069,Y -486.115,Z 683.524,A 0.000,B 0.000,C 90.000,E1 274.245} C_DIS
LIN {X -0.227,Y -487.038,Z 683.521,A 0.000,B 0.000,C 90.000,E1 273.784} C_DIS
LIN {X -0.062,Y -487.588,Z 683.518,A 0.000,B 0.000,C 90.000,E1 273.269} C_DIS
LIN {X 0.136,Y -487.825,Z 683.515,A 0.000,B 0.000,C 90.000,E1 272.751} C_DIS
LIN {X -0.173,Y -487.751,Z 683.513,A 0.000,B 0.000,C 90.000,E1 272.293} C_DIS
LIN {X 0.023,Y -487.352,Z 683.510,A 0.000,B 0.000,C 90.000,E1 271.776} C_DIS
LIN {X 0.202,Y -486.601,Z 683.507,A 0.000,B 0.000,C 90.000,E1 271.260} C_DIS
LIN {X -0.106,Y -485.461,Z 683.504,A 0.000,B 0.000,C 90.000,E1 270.802} C_DIS
LIN {X 0.069,Y -483.822,Z 683.502,A 0.000,B 0.000,C 90.000,E1 270.286} C_DIS
LIN {X 0.235,Y -481.628,Z 683.499,A 0.000,B 0.000,C 90.000,E1 269.771} C_DIS
LIN {X -0.093,Y -478.694,Z 683.496,A 0.000,B 0.000,C 90.000,E1 269.312} C_DIS
LIN {X 0.042,Y -474.987,Z 683.493,A 0.000,B 0.000,C 90.000,E1 268.797} C_DIS
LIN {X -0.138,Y -472.796,Z 683.492,A 0.000,B 0.000,C 90.000,E1 268.568} C_DIS
LIN {X 0.018,Y -467.568,Z 683.489,A 0.000,B 0.000,C 90.000,E1 268.051} C_DIS
LIN {X -0.007,Y -461.504,Z 683.487,A 0.000,B 0.000,C 90.000,E1 267.593} C_DIS
LIN {X 0.055,Y -454.838,Z 683.484,A 0.000,B 0.000,C 90.000,E1 267.192} C_DIS
LIN {X 0.203,Y -447.771,Z 683.483,A 0.000,B 0.000,C 90.000,E1 266.849} C_DIS
LIN {X -0.027,Y -440.452,Z 683.481,A 0.000,B 0.000,C 90.000,E1 266.617} C_DIS
LIN {X 0.167,Y -432.355,Z 683.480,A 0.000,B 0.000,C 90.000,E1 266.388} C_DIS
LIN {X 0.035,Y -423.189,Z 683.479,A 0.000,B 0.000,C 90.000,E1 266.274} C_DIS
LIN {X 0.117,Y -415.744,Z 683.479,A 0.000,B 0.000,C 90.000,E1 266.216} C_DIS
LIN {X 0.026,Y -180.931,Z 683.479,A 0.000,B 0.000,C 90.000,E1 266.216} C_DIS
LIN {X -0.078,Y -180.766,Z 683.471,A 0.000,B 0.000,C 90.000,E1 264.723} C_DIS
LIN {X -0.040,Y -178.985,Z 683.444,A 0.000,B 0.000,C 90.000,E1 259.982} C_DIS
LIN {X -0.029,Y -177.962,Z 683.435,A 0.000,B 0.000,C 90.000,E1 258.285} C_DIS
LIN {X -0.010,Y -175.603,Z 683.411,A 0.000,B 0.000,C 90.000,E1 254.031} C_DIS
LIN {X 0.003,Y -172.327,Z 683.388,A 0.000,B 0.000,C 90.000,E1 249.752} C_DIS
LIN {X -0.019,Y -171.804,Z 683.383,A 0.000,B 0.000,C 90.000,E1 248.901} C_DIS
LIN {X -0.011,Y -170.263,Z 683.373,A 0.000,B 0.000,C 90.000,E1 247.177} C_DIS
LIN {X -0.074,Y -166.806,Z 683.349,A 0.000,B 0.000,C 90.000,E1 242.871} C_DIS
LIN {X 0.069,Y -162.787,Z 683.325,A 0.000,B 0.000,C 90.000,E1 238.456} C_DIS
LIN {X 0.044,Y -161.475,Z 683.315,A 0.000,B 0.000,C 90.000,E1 236.707} C_DIS
LIN {X 0.085,Y -157.470,Z 683.291,A 0.000,B 0.000,C 90.000,E1 232.271} C_DIS
LIN {X 0.017,Y -155.484,Z 683.276,A 0.000,B 0.000,C 90.000,E1 229.622} C_DIS
LIN {X -0.050,Y -151.793,Z 683.251,A 0.000,B 0.000,C 90.000,E1 225.162} C_DIS
LIN {X -0.037,Y -150.001,Z 683.236,A 0.000,B 0.000,C 90.000,E1 222.447} C_DIS
LIN {X -0.006,Y -146.829,Z 683.211,A 0.000,B 0.000,C 90.000,E1 217.890} C_DIS
LIN {X -0.019,Y -145.410,Z 683.195,A 0.000,B 0.000,C 90.000,E1 215.152} C_DIS
LIN {X 0.017,Y -142.841,Z 683.170,A 0.000,B 0.000,C 90.000,E1 210.541} C_DIS
LIN {X -0.053,Y -141.454,Z 683.149,A 0.000,B 0.000,C 90.000,E1 206.873} C_DIS
LIN {X -0.013,Y -139.372,Z 683.113,A 0.000,B 0.000,C 90.000,E1 200.355} C_DIS
LIN {X -0.071,Y -138.822,Z 683.098,A 0.000,B 0.000,C 90.000,E1 197.583} C_DIS
LIN {X 0.017,Y -138.352,Z 683.056,A 0.000,B 0.000,C 90.000,E1 190.074} C_DIS
LIN {X -0.010,Y -139.533,Z 683.004,A 0.000,B 0.000,C 90.000,E1 180.745} C_DIS
LIN {X -0.057,Y -141.215,Z 682.973,A 0.000,B 0.000,C 90.000,E1 175.179} C_DIS
LIN {X 0.043,Y -142.588,Z 682.958,A 0.000,B 0.000,C 90.000,E1 172.356} C_DIS
LIN {X -0.004,Y -144.888,Z 682.932,A 0.000,B 0.000,C 90.000,E1 167.757} C_DIS
LIN {X -0.050,Y -147.516,Z 682.912,A 0.000,B 0.000,C 90.000,E1 164.102} C_DIS
LIN {X 0.025,Y -150.110,Z 682.891,A 0.000,B 0.000,C 90.000,E1 160.423} C_DIS
LIN {X 0.037,Y -153.469,Z 682.871,A 0.000,B 0.000,C 90.000,E1 156.794} C_DIS
LIN {X 0.027,Y -157.832,Z 682.846,A 0.000,B 0.000,C 90.000,E1 152.308} C_DIS
LIN {X 0.058,Y -162.117,Z 682.826,A 0.000,B 0.000,C 90.000,E1 148.742} C_DIS
LIN {X -0.057,Y -166.318,Z 682.807,A 0.000,B 0.000,C 90.000,E1 145.261} C_DIS
LIN {X 0.045,Y -171.336,Z 682.788,A 0.000,B 0.000,C 90.000,E1 141.743} C_DIS
LIN {X -0.027,Y -176.238,Z 682.768,A 0.000,B 0.000,C 90.000,E1 138.324} C_DIS
LIN {X 0.092,Y -180.518,Z 682.754,A 0.000,B 0.000,C 90.000,E1 135.729} C_DIS
LIN {X 0.072,Y -185.921,Z 682.735,A 0.000,B 0.000,C 90.000,E1 132.366} C_DIS
LIN {X 0.036,Y -191.169,Z 682.720,A 0.000,B 0.000,C 90.000,E1 129.519} C_DIS
LIN {X 0.019,Y -288.980,Z 682.720,A 0.000,B 0.000,C 90.000,E1 129.519} C_DIS
LIN {X -0.006,Y -291.289,Z 682.719,A 0.000,B 0.000,C 90.000,E1 129.483} C_DIS
LIN {X -0.032,Y -295.456,Z 682.718,A 0.000,B 0.000,C 90.000,E1 129.277} C_DIS
LIN {X -0.057,Y -297.864,Z 682.717,A 0.000,B 0.000,C 90.000,E1 129.072} C_DIS
LIN {X 0.041,Y -301.690,Z 682.714,A 0.000,B 0.000,C 90.000,E1 128.543} C_DIS
LIN {X -0.014,Y -303.421,Z 682.712,A 0.000,B 0.000,C 90.000,E1 128.222} C_DIS
LIN {X -0.017,Y -304.777,Z 682.711,A 0.000,B 0.000,C 90.000,E1 127.890} C_DIS
LIN {X -0.055,Y -308.558,Z 682.703,A 0.000,B 0.000,C 90.000,E1 126.583} C_DIS
LIN {X 0.197,Y -318.578,Z 682.685,A 0.000,B 0.000,C 90.000,E1 123.293} C_DIS
LIN {X -0.007,Y -328.911,Z 682.669,A 0.000,B 0.000,C 90.000,E1 120.463} C_DIS
LIN {X 0.030,Y -340.595,Z 682.654,A 0.000,B 0.000,C 90.000,E1 117.641} C_DIS
LIN {X -0.066,Y -353.729,Z 682.638,A 0.000,B 0.000,C 90.000,E1 114.899} C_DIS
LIN {X 0.173,Y -366.721,Z 682.625,A 0.000,B 0.000,C 90.000,E1 112.461} C_DIS
LIN {X 0.125,Y -381.047,Z 682.612,A 0.000,B 0.000,C 90.000,E1 110.120} C_DIS
LIN {X 0.172,Y -396.811,Z 682.599,A 0.000,B 0.000,C 90.000,E1 107.819} C_DIS
LIN {X -0.013,Y -414.128,Z 682.587,A 0.000,B 0.000,C 90.000,E1 105.607} C_DIS
LIN {X 0.118,Y -433.113,Z 682.575,A 0.000,B 0.000,C 90.000,E1 103.411} C_DIS
LIN {X 0.091,Y -453.204,Z 682.563,A 0.000,B 0.000,C 90.000,E1 101.366} C_DIS
LIN {X -0.068,Y -468.636,Z 682.555,A 0.000,B 0.000,C 90.000,E1 99.962} C_DIS
LIN {X -0.021,Y -470.839,Z 682.554,A 0.000,B 0.000,C 90.000,E1 99.726} C_DIS
LIN {X -0.249,Y -472.655,Z 682.553,A 0.000,B 0.000,C 90.000,E1 99.500} C_DIS
LIN {X 0.067,Y -474.019,Z 682.551,A 0.000,B 0.000,C 90.000,E1 99.208} C_DIS
LIN {X 0.183,Y -475.733,Z 682.548,A 0.000,B 0.000,C 90.000,E1 98.690} C_DIS
LIN {X -0.093,Y -476.374,Z 682.546,A 0.000,B 0.000,C 90.000,E1 98.219} C_DIS
LIN {X 0.042,Y -476.048,Z 682.543,A 0.000,B 0.000,C 90.000,E1 97.701} C_DIS
LIN {X 0.181,Y -474.706,Z 682.540,A 0.000,B 0.000,C 90.000,E1 97.182} C_DIS
LIN {X 0.044,Y -473.590,Z 682.539,A 0.000,B 0.000,C 90.000,E1 96.947} C_DIS
LIN {X 0.172,Y -470.378,Z 682.536,A 0.000,B 0.000,C 90.000,E1 96.429} C_DIS
LIN {X 0.026,Y -453.755,Z 682.522,A 0.000,B 0.000,C 90.000,E1 93.898} C_DIS
LIN {X 0.001,Y -437.593,Z 682.506,A 0.000,B 0.000,C 90.000,E1 91.031} C_DIS
LIN {X -0.068,Y -430.251,Z 682.498,A 0.000,B 0.000,C 90.000,E1 89.714} C_DIS
LIN {X -0.107,Y -421.006,Z 682.489,A 0.000,B 0.000,C 90.000,E1 88.108} C_DIS
LIN {X -0.111,Y -408.539,Z 682.477,A 0.000,B 0.000,C 90.000,E1 85.927} C_DIS
LIN {X 0.086,Y -394.509,Z 682.463,A 0.000,B 0.000,C 90.000,E1 83.394} C_DIS
LIN {X -0.009,Y -380.960,Z 682.449,A 0.000,B 0.000,C 90.000,E1 80.849} C_DIS
LIN {X 0.036,Y -369.297,Z 682.436,A 0.000,B 0.000,C 90.000,E1 78.522} C_DIS
LIN {X -0.052,Y -355.316,Z 682.420,A 0.000,B 0.000,C 90.000,E1 75.574} C_DIS
LIN {X -0.043,Y -343.264,Z 682.405,A 0.000,B 0.000,C 90.000,E1 72.851} C_DIS
LIN {X 0.031,Y -331.767,Z 682.389,A 0.000,B 0.000,C 90.000,E1 70.061} C_DIS
LIN {X -0.137,Y -317.695,Z 682.368,A 0.000,B 0.000,C 90.000,E1 66.305} C_DIS
LIN {X -0.042,Y -306.390,Z 682.349,A 0.000,B 0.000,C 90.000,E1 62.743} C_DIS
LIN {X -0.029,Y -297.107,Z 682.330,A 0.000,B 0.000,C 90.000,E1 59.459} C_DIS
LIN {X 0.147,Y -288.526,Z 682.312,A 0.000,B 0.000,C 90.000,E1 56.087} C_DIS
LIN {X 0.099,Y -283.572,Z 682.300,A 0.000,B 0.000,C 90.000,E1 54.069} C_DIS
LIN {X 0.069,Y -278.598,Z 682.289,A 0.000,B 0.000,C 90.000,E1 52.029} C_DIS
LIN {X -0.050,Y -273.399,Z 682.278,A 0.000,B 0.000,C 90.000,E1 49.989} C_DIS
LIN {X -0.087,Y -269.785,Z 682.270,A 0.000,B 0.000,C 90.000,E1 48.609} C_DIS
LIN {X -0.041,Y -263.977,Z 682.258,A 0.000,B 0.000,C 90.000,E1 46.500} C_DIS
LIN {X 0.072,Y -257.941,Z 682.246,A 0.000,B 0.000,C 90.000,E1 44.352} C_DIS
LIN {X 0.066,Y -251.779,Z 682.235,A 0.000,B 0.000,C 90.000,E1 42.204} C_DIS
LIN {X 0.145,Y -245.492,Z 682.222,A 0.000,B 0.000,C 90.000,E1 40.011} C_DIS
LIN {X -0.073,Y -235.182,Z 682.202,A 0.000,B 0.000,C 90.000,E1 36.377} C_DIS
LIN {X -0.065,Y -227.501,Z 682.185,A 0.000,B 0.000,C 90.000,E1 33.372} C_DIS
LIN {X -0.116,Y -220.649,Z 682.168,A 0.000,B 0.000,C 90.000,E1 30.335} C_DIS
LIN {X 0.015,Y -214.590,Z 682.151,A 0.000,B 0.000,C 90.000,E1 27.206} C_DIS
LIN {X -0.010,Y -209.306,Z 682.134,A 0.000,B 0.000,C 90.000,E1 24.079} C_DIS
LIN {X -0.035,Y -203.931,Z 682.112,A 0.000,B 0.000,C 90.000,E1 20.120} C_DIS
LIN {X 0.072,Y -199.679,Z 682.089,A 0.000,B 0.000,C 90.000,E1 16.079} C_DIS
LIN {X -0.007,Y -195.996,Z 682.062,A 0.000,B 0.000,C 90.000,E1 11.243} C_DIS
LIN {X 0.022,Y -193.308,Z 682.026,A 0.000,B 0.000,C 90.000,E1 4.702} C_DIS
LIN {X -0.013,Y -194.582,Z 681.966,A 0.000,B 0.000,C 90.000,E1 353.799} C_DIS
LIN {X -0.068,Y -198.082,Z 681.934,A 0.000,B 0.000,C 90.000,E1 348.105} C_DIS
LIN {X 0.023,Y -201.815,Z 681.911,A 0.000,B 0.000,C 90.000,E1 344.031} C_DIS
LIN {X 0.061,Y -206.497,Z 681.889,A 0.000,B 0.000,C 90.000,E1 340.007} C_DIS
LIN {X 0.012,Y -211.985,Z 681.867,A 0.000,B 0.000,C 90.000,E1 336.049} C_DIS
LIN {X -0.092,Y -218.208,Z 681.845,A 0.000,B 0.000,C 90.000,E1 332.153} C_DIS
LIN {X 0.033,Y -225.197,Z 681.824,A 0.000,B 0.000,C 90.000,E1 328.250} C_DIS
LIN {X -0.152,Y -232.702,Z 681.802,A 0.000,B 0.000,C 90.000,E1 324.482} C_DIS
LIN {X 0.053,Y -240.933,Z 681.782,A 0.000,B 0.000,C 90.000,E1 320.678} C_DIS
LIN {X 0.062,Y -249.950,Z 681.761,A 0.000,B 0.000,C 90.000,E1 316.986} C_DIS
LIN {X 0.010,Y -260.187,Z 681.741,A 0.000,B 0.000,C 90.000,E1 313.380} C_DIS
LIN {X 0.086,Y -270.272,Z 681.723,A 0.000,B 0.000,C 90.000,E1 310.172} C_DIS
LIN {X -0.070,Y -281.594,Z 681.706,A 0.000,B 0.000,C 90.000,E1 307.076} C_DIS
LIN {X 0.037,Y -295.539,Z 681.687,A 0.000,B 0.000,C 90.000,E1 303.658} C_DIS
LIN {X 0.119,Y -310.781,Z 681.669,A 0.000,B 0.000,C 90.000,E1 300.335} C_DIS
LIN {X 0.061,Y -327.687,Z 681.651,A 0.000,B 0.000,C 90.000,E1 297.129} C_DIS
LIN {X -0.057,Y -343.873,Z 681.635,A 0.000,B 0.000,C 90.000,E1 294.335} C_DIS
LIN {X 0.107,Y -364.783,Z 681.617,A 0.000,B 0.000,C 90.000,E1 290.972} C_DIS
LIN {X 0.018,Y -377.163,Z 681.607,A 0.000,B 0.000,C 90.000,E1 289.214} C_DIS
LIN {X -0.123,Y -402.261,Z 681.589,A 0.000,B 0.000,C 90.000,E1 286.079} C_DIS
LIN {X -0.065,Y -411.555,Z 681.583,A 0.000,B 0.000,C 90.000,E1 284.954} C_DIS
LIN {X -0.165,Y -422.920,Z 681.575,A 0.000,B 0.000,C 90.000,E1 283.592} C_DIS
LIN {X -0.189,Y -433.799,Z 681.568,A 0.000,B 0.000,C 90.000,E1 282.243} C_DIS
LIN {X 0.167,Y -442.048,Z 681.562,A 0.000,B 0.000,C 90.000,E1 281.130} C_DIS
LIN {X -0.040,Y -459.919,Z 681.549,A 0.000,B 0.000,C 90.000,E1 278.803} C_DIS
LIN {X 0.110,Y -467.962,Z 681.543,A 0.000,B 0.000,C 90.000,E1 277.757} C_DIS
LIN {X 0.035,Y -473.472,Z 681.539,A 0.000,B 0.000,C 90.000,E1 277.004} C_DIS
LIN {X -0.056,Y -478.161,Z 681.535,A 0.000,B 0.000,C 90.000,E1 276.258} C_DIS
LIN {X 0.088,Y -480.754,Z 681.532,A 0.000,B 0.000,C 90.000,E1 275.739} C_DIS
LIN {X 0.247,Y -482.881,Z 681.529,A 0.000,B 0.000,C 90.000,E1 275.220} C_DIS
LIN {X -0.062,Y -484.621,Z 681.526,A 0.000,B 0.000,C 90.000,E1 274.759} C_DIS
LIN {X 0.078,Y -485.929,Z 681.524,A 0.000,B 0.000,C 90.000,E1 274.245} C_DIS
LIN {X -0.220,Y -486.861,Z 681.521,A 0.000,B 0.000,C 90.000,E1 273.784} C_DIS
LIN {X -0.056,Y -487.430,Z 681.518,A 0.000,B 0.000,C 90.000,E1 273.269} C_DIS
LIN {X 0.142,Y -487.701,Z 681.515,A 0.000,B 0.000,C 90.000,E1 272.751} C_DIS
LIN {X -0.169,Y -487.645,Z 681.513,A 0.000,B 0.000,C 90.000,E1 272.293} C_DIS
LIN {X 0.027,Y -487.291,Z 681.510,A 0.000,B 0.000,C 90.000,E1 271.776} C_DIS
LIN {X 0.205,Y -486.573,Z 681.507,A 0.000,B 0.000,C 90.000,E1 271.260} C_DIS
LIN {X -0.103,Y -485.429,Z 681.504,A 0.000,B 0.000,C 90.000,E1 270.802} C_DIS
LIN {X 0.071,Y -483.791,Z 681.502,A 0.000,B 0.000,C 90.000,E1 270.286} C_DIS
LIN {X -0.087,Y -482.815,Z 681.500,A 0.000,B 0.000,C 90.000,E1 270.057} C_DIS
LIN {X 0.073,Y -480.287,Z 681.497,A 0.000,B 0.000,C 90.000,E1 269.542} C_DIS
LIN {X 0.216,Y -476.983,Z 681.495,A 0.000,B 0.000,C 90.000,E1 269.026} C_DIS
LIN {X -0.134,Y -472.783,Z 681.492,A 0.000,B 0.000,C 90.000,E1 268.568} C_DIS
LIN {X 0.157,Y -470.350,Z 681.491,A 0.000,B 0.000,C 90.000,E1 268.282} C_DIS
LIN {X -0.192,Y -464.354,Z 681.488,A 0.000,B 0.000,C 90.000,E1 267.822} C_DIS
LIN {X -0.084,Y -461.365,Z 681.487,A 0.000,B 0.000,C 90.000,E1 267.593} C_DIS
LIN {X -0.032,Y -454.665,Z 681.484,A 0.000,B 0.000,C 90.000,E1 267.192} C_DIS
LIN {X 0.115,Y -447.624,Z 681.483,A 0.000,B 0.000,C 90.000,E1 266.849} C_DIS
LIN {X -0.107,Y -440.172,Z 681.481,A 0.000,B 0.000,C 90.000,E1 266.617} C_DIS
LIN {X 0.120,Y -432.165,Z 681.480,A 0.000,B 0.000,C 90.000,E1 266.388} C_DIS
LIN {X 0.006,Y -423.206,Z 681.479,A 0.000,B 0.000,C 90.000,E1 266.274} C_DIS
LIN {X 0.081,Y -416.174,Z 681.479,A 0.000,B 0.000,C 90.000,E1 266.216} C_DIS
LIN {X 0.010,Y -180.931,Z 681.479,A 0.000,B 0.000,C 90.000,E1 266.216} C_DIS
LIN {X 0.085,Y -180.764,Z 681.471,A 0.000,B 0.000,C 90.000,E1 264.666} C_DIS
LIN {X -0.058,Y -178.983,Z 681.444,A 0.000,B 0.000,C 90.000,E1 259.982} C_DIS
LIN {X -0.045,Y -177.957,Z 681.435,A 0.000,B 0.000,C 90.000,E1 258.285} C_DIS
LIN {X -0.027,Y -175.600,Z 681.411,A 0.000,B 0.000,C 90.000,E1 254.031} C_DIS
LIN {X -0.014,Y -172.323,Z 681.388,A 0.000,B 0.000,C 90.000,E1 249.752} C_DIS
LIN {X -0.035,Y -171.800,Z 681.383,A 0.000,B 0.000,C 90.000,E1 248.901} C_DIS
LIN {X 0.002,Y -169.474,Z 681.368,A 0.000,B 0.000,C 90.000,E1 246.305} C_DIS
LIN {X -0.091,Y -166.801,Z 681.349,A 0.000,B 0.000,C 90.000,E1 242.871} C_DIS
LIN {X 0.052,Y -162.782,Z 681.325,A 0.000,B 0.000,C 90.000,E1 238.456} C_DIS
LIN {X 0.028,Y -161.471,Z 681.315,A 0.000,B 0.000,C 90.000,E1 236.707} C_DIS
LIN {X 0.068,Y -157.465,Z 681.291,A 0.000,B 0.000,C 90.000,E1 232.271} C_DIS
LIN {X 0.002,Y -155.480,Z 681.276,A 0.000,B 0.000,C 90.000,E1 229.622} C_DIS
LIN {X -0.065,Y -151.789,Z 681.251,A 0.000,B 0.000,C 90.000,E1 225.162} C_DIS
LIN {X -0.053,Y -149.996,Z 681.236,A 0.000,B 0.000,C 90.000,E1 222.447} C_DIS
LIN {X -0.022,Y -146.826,Z 681.210,A 0.000,B 0.000,C 90.000,E1 217.890} C_DIS
LIN {X -0.034,Y -145.406,Z 681.195,A 0.000,B 0.000,C 90.000,E1 215.152} C_DIS
LIN {X 0.002,Y -142.837,Z 681.170,A 0.000,B 0.000,C 90.000,E1 210.541} C_DIS
LIN {X -0.068,Y -141.451,Z 681.149,A 0.000,B 0.000,C 90.000,E1 206.873} C_DIS
LIN {X -0.028,Y -139.372,Z 681.113,A 0.000,B 0.000,C 90.000,E1 200.355} C_DIS
LIN {X 0.046,Y -138.821,Z 681.097,A 0.000,B 0.000,C 90.000,E1 197.528} C_DIS
LIN {X 0.003,Y -138.353,Z 681.056,A 0.000,B 0.000,C 90.000,E1 190.074} C_DIS
LIN {X -0.024,Y -139.533,Z 681.004,A 0.000,B 0.000,C 90.000,E1 180.745} C_DIS
LIN {X 0.069,Y -141.218,Z 680.973,A 0.000,B 0.000,C 90.000,E1 175.122} C_DIS
LIN {X 0.028,Y -142.591,Z 680.958,A 0.000,B 0.000,C 90.000,E1 172.356} C_DIS
LIN {X -0.018,Y -144.892,Z 680.932,A 0.000,B 0.000,C 90.000,E1 167.757} C_DIS
LIN {X -0.065,Y -147.519,Z 680.912,A 0.000,B 0.000,C 90.000,E1 164.102} C_DIS
LIN {X 0.009,Y -150.114,Z 680.891,A 0.000,B 0.000,C 90.000,E1 160.423} C_DIS
LIN {X 0.021,Y -153.475,Z 680.871,A 0.000,B 0.000,C 90.000,E1 156.794} C_DIS
LIN {X 0.085,Y -157.839,Z 680.846,A 0.000,B 0.000,C 90.000,E1 152.281} C_DIS
LIN {X 0.042,Y -162.123,Z 680.826,A 0.000,B 0.000,C 90.000,E1 148.742} C_DIS
LIN {X -0.074,Y -166.326,Z 680.807,A 0.000,B 0.000,C 90.000,E1 145.261} C_DIS
LIN {X 0.028,Y -171.343,Z 680.788,A 0.000,B 0.000,C 90.000,E1 141.743} C_DIS
LIN {X -0.045,Y -176.247,Z 680.768,A 0.000,B 0.000,C 90.000,E1 138.324} C_DIS
LIN {X 0.074,Y -180.528,Z 680.754,A 0.000,B 0.000,C 90.000,E1 135.729} C_DIS
LIN {X 0.054,Y -185.930,Z 680.735,A 0.000,B 0.000,C 90.000,E1 132.366} C_DIS
LIN {X -0.082,Y -191.155,Z 680.720,A 0.000,B 0.000,C 90.000,E1 129.564} C_DIS
LIN {X -0.160,Y -289.242,Z 680.720,A 0.000,B 0.000,C 90.000,E1 129.564} C_DIS
LIN {X -0.032,Y -291.758,Z 680.719,A 0.000,B 0.000,C 90.000,E1 129.483} C_DIS
LIN {X -0.059,Y -295.629,Z 680.718,A 0.000,B 0.000,C 90.000,E1 129.277} C_DIS
LIN {X 0.103,Y -297.974,Z 680.717,A 0.000,B 0.000,C 90.000,E1 129.036} C_DIS
LIN {X -0.048,Y -301.803,Z 680.714,A 0.000,B 0.000,C 90.000,E1 128.543} C_DIS
LIN {X 0.137,Y -303.497,Z 680.712,A 0.000,B 0.000,C 90.000,E1 128.177} C_DIS
LIN {X -0.106,Y -304.827,Z 680.710,A 0.000,B 0.000,C 90.000,E1 127.890} C_DIS
LIN {X 0.108,Y -312.420,Z 680.696,A 0.000,B 0.000,C 90.000,E1 125.231} C_DIS
LIN {X 0.147,Y -323.048,Z 680.678,A 0.000,B 0.000,C 90.000,E1 122.005} C_DIS
LIN {X -0.102,Y -333.975,Z 680.662,A 0.000,B 0.000,C 90.000,E1 119.205} C_DIS
LIN {X -0.085,Y -346.300,Z 680.647,A 0.000,B 0.000,C 90.000,E1 116.411} C_DIS
LIN {X 0.150,Y -360.125,Z 680.631,A 0.000,B 0.000,C 90.000,E1 113.643} C_DIS
LIN {X 0.074,Y -373.781,Z 680.618,A 0.000,B 0.000,C 90.000,E1 111.280} C_DIS
LIN {X 0.061,Y -388.822,Z 680.605,A 0.000,B 0.000,C 90.000,E1 108.960} C_DIS
LIN {X 0.177,Y -405.357,Z 680.593,A 0.000,B 0.000,C 90.000,E1 106.677} C_DIS
LIN {X 0.090,Y -423.507,Z 680.581,A 0.000,B 0.000,C 90.000,E1 104.481} C_DIS
LIN {X 0.086,Y -443.191,Z 680.569,A 0.000,B 0.000,C 90.000,E1 102.355} C_DIS
LIN {X -0.142,Y -463.570,Z 680.558,A 0.000,B 0.000,C 90.000,E1 100.423} C_DIS
LIN {X -0.171,Y -468.747,Z 680.555,A 0.000,B 0.000,C 90.000,E1 99.962} C_DIS
LIN {X -0.122,Y -470.939,Z 680.554,A 0.000,B 0.000,C 90.000,E1 99.726} C_DIS
LIN {X 0.115,Y -472.749,Z 680.553,A 0.000,B 0.000,C 90.000,E1 99.443} C_DIS
LIN {X -0.034,Y -474.107,Z 680.551,A 0.000,B 0.000,C 90.000,E1 99.208} C_DIS
LIN {X 0.082,Y -475.814,Z 680.548,A 0.000,B 0.000,C 90.000,E1 98.690} C_DIS
LIN {X -0.194,Y -476.448,Z 680.546,A 0.000,B 0.000,C 90.000,E1 98.219} C_DIS
LIN {X -0.059,Y -476.115,Z 680.543,A 0.000,B 0.000,C 90.000,E1 97.701} C_DIS
LIN {X 0.082,Y -474.767,Z 680.540,A 0.000,B 0.000,C 90.000,E1 97.182} C_DIS
LIN {X -0.056,Y -473.645,Z 680.539,A 0.000,B 0.000,C 90.000,E1 96.947} C_DIS
LIN {X 0.074,Y -470.430,Z 680.536,A 0.000,B 0.000,C 90.000,E1 96.429} C_DIS
LIN {X -0.068,Y -453.781,Z 680.522,A 0.000,B 0.000,C 90.000,E1 93.898} C_DIS
LIN {X 0.078,Y -436.166,Z 680.504,A 0.000,B 0.000,C 90.000,E1 90.745} C_DIS
LIN {X -0.007,Y -428.789,Z 680.497,A 0.000,B 0.000,C 90.000,E1 89.427} C_DIS
LIN {X -0.073,Y -419.483,Z 680.488,A 0.000,B 0.000,C 90.000,E1 87.822} C_DIS
LIN {X -0.119,Y -407.011,Z 680.476,A 0.000,B 0.000,C 90.000,E1 85.641} C_DIS
LIN {X 0.025,Y -393.022,Z 680.462,A 0.000,B 0.000,C 90.000,E1 83.109} C_DIS
LIN {X -0.051,Y -379.567,Z 680.448,A 0.000,B 0.000,C 90.000,E1 80.557} C_DIS
LIN {X -0.049,Y -366.557,Z 680.433,A 0.000,B 0.000,C 90.000,E1 77.937} C_DIS
LIN {X 0.156,Y -351.370,Z 680.415,A 0.000,B 0.000,C 90.000,E1 74.629} C_DIS
LIN {X 0.139,Y -338.235,Z 680.398,A 0.000,B 0.000,C 90.000,E1 71.583} C_DIS
LIN {X 0.076,Y -323.539,Z 680.377,A 0.000,B 0.000,C 90.000,E1 67.847} C_DIS
LIN {X 0.026,Y -312.568,Z 680.359,A 0.000,B 0.000,C 90.000,E1 64.665} C_DIS
LIN {X -0.066,Y -302.791,Z 680.341,A 0.000,B 0.000,C 90.000,E1 61.435} C_DIS
LIN {X -0.013,Y -293.835,Z 680.323,A 0.000,B 0.000,C 90.000,E1 58.122} C_DIS
LIN {X -0.145,Y -287.119,Z 680.308,A 0.000,B 0.000,C 90.000,E1 55.468} C_DIS
LIN {X 0.035,Y -280.533,Z 680.293,A 0.000,B 0.000,C 90.000,E1 52.718} C_DIS
LIN {X 0.121,Y -275.405,Z 680.281,A 0.000,B 0.000,C 90.000,E1 50.642} C_DIS
LIN {X -0.092,Y -270.039,Z 680.270,A 0.000,B 0.000,C 90.000,E1 48.609} C_DIS
LIN {X -0.042,Y -264.240,Z 680.258,A 0.000,B 0.000,C 90.000,E1 46.500} C_DIS
LIN {X 0.077,Y -258.181,Z 680.247,A 0.000,B 0.000,C 90.000,E1 44.352} C_DIS
LIN {X 0.075,Y -252.009,Z 680.235,A 0.000,B 0.000,C 90.000,E1 42.204} C_DIS
LIN {X 0.159,Y -245.690,Z 680.222,A 0.000,B 0.000,C 90.000,E1 40.011} C_DIS
LIN {X -0.054,Y -235.375,Z 680.202,A 0.000,B 0.000,C 90.000,E1 36.377} C_DIS
LIN {X -0.043,Y -227.688,Z 680.185,A 0.000,B 0.000,C 90.000,E1 33.372} C_DIS
LIN {X -0.090,Y -220.832,Z 680.168,A 0.000,B 0.000,C 90.000,E1 30.335} C_DIS
LIN {X 0.047,Y -214.781,Z 680.151,A 0.000,B 0.000,C 90.000,E1 27.206} C_DIS
LIN {X 0.025,Y -209.492,Z 680.134,A 0.000,B 0.000,C 90.000,E1 24.079} C_DIS
LIN {X 0.003,Y -204.099,Z 680.112,A 0.000,B 0.000,C 90.000,E1 20.120} C_DIS
LIN {X -0.078,Y -199.832,Z 680.090,A 0.000,B 0.000,C 90.000,E1 16.134} C_DIS
LIN {X 0.041,Y -196.147,Z 680.063,A 0.000,B 0.000,C 90.000,E1 11.243} C_DIS
LIN {X 0.076,Y -193.437,Z 680.026,A 0.000,B 0.000,C 90.000,E1 4.702} C_DIS
LIN {X -0.008,Y -194.671,Z 679.966,A 0.000,B 0.000,C 90.000,E1 353.799} C_DIS
LIN {X 0.107,Y -197.546,Z 679.938,A 0.000,B 0.000,C 90.000,E1 348.870} C_DIS
LIN {X -0.064,Y -201.058,Z 679.916,A 0.000,B 0.000,C 90.000,E1 344.866} C_DIS
LIN {X -0.113,Y -205.553,Z 679.893,A 0.000,B 0.000,C 90.000,E1 340.859} C_DIS
LIN {X 0.002,Y -210.884,Z 679.871,A 0.000,B 0.000,C 90.000,E1 336.847} C_DIS
LIN {X -0.031,Y -216.937,Z 679.850,A 0.000,B 0.000,C 90.000,E1 332.922} C_DIS
LIN {X 0.141,Y -223.788,Z 679.828,A 0.000,B 0.000,C 90.000,E1 328.997} C_DIS
LIN {X 0.106,Y -231.178,Z 679.807,A 0.000,B 0.000,C 90.000,E1 325.182} C_DIS
LIN {X -0.060,Y -239.222,Z 679.786,A 0.000,B 0.000,C 90.000,E1 321.457} C_DIS
LIN {X 0.104,Y -248.058,Z 679.765,A 0.000,B 0.000,C 90.000,E1 317.715} C_DIS
LIN {X 0.144,Y -257.030,Z 679.747,A 0.000,B 0.000,C 90.000,E1 314.433} C_DIS
LIN {X -0.026,Y -267.925,Z 679.727,A 0.000,B 0.000,C 90.000,E1 310.906} C_DIS
LIN {X 0.135,Y -278.937,Z 679.710,A 0.000,B 0.000,C 90.000,E1 307.729} C_DIS
LIN {X 0.090,Y -292.639,Z 679.691,A 0.000,B 0.000,C 90.000,E1 304.326} C_DIS
LIN {X 0.073,Y -307.605,Z 679.672,A 0.000,B 0.000,C 90.000,E1 301.003} C_DIS
LIN {X 0.065,Y -324.194,Z 679.654,A 0.000,B 0.000,C 90.000,E1 297.769} C_DIS
LIN {X -0.141,Y -338.336,Z 679.640,A 0.000,B 0.000,C 90.000,E1 295.283} C_DIS
LIN {X -0.144,Y -353.076,Z 679.627,A 0.000,B 0.000,C 90.000,E1 292.823} C_DIS
LIN {X -0.024,Y -372.775,Z 679.610,A 0.000,B 0.000,C 90.000,E1 289.812} C_DIS
LIN {X 0.190,Y -390.431,Z 679.597,A 0.000,B 0.000,C 90.000,E1 287.457} C_DIS
LIN {X 0.166,Y -406.837,Z 679.586,A 0.000,B 0.000,C 90.000,E1 285.481} C_DIS
LIN {X 0.134,Y -420.536,Z 679.577,A 0.000,B 0.000,C 90.000,E1 283.828} C_DIS
LIN {X 0.075,Y -431.508,Z 679.569,A 0.000,B 0.000,C 90.000,E1 282.479} C_DIS
LIN {X -0.023,Y -439.888,Z 679.563,A 0.000,B 0.000,C 90.000,E1 281.422} C_DIS
LIN {X -0.077,Y -451.702,Z 679.555,A 0.000,B 0.000,C 90.000,E1 279.849} C_DIS
LIN {X -0.165,Y -465.786,Z 679.545,A 0.000,B 0.000,C 90.000,E1 278.049} C_DIS
LIN {X 0.202,Y -471.521,Z 679.540,A 0.000,B 0.000,C 90.000,E1 277.239} C_DIS
LIN {X 0.159,Y -476.501,Z 679.536,A 0.000,B 0.000,C 90.000,E1 276.486} C_DIS
LIN {X -0.185,Y -479.322,Z 679.533,A 0.000,B 0.000,C 90.000,E1 276.024} C_DIS
LIN {X -0.085,Y -481.693,Z 679.531,A 0.000,B 0.000,C 90.000,E1 275.511} C_DIS
LIN {X -0.053,Y -484.471,Z 679.526,A 0.000,B 0.000,C 90.000,E1 274.759} C_DIS
LIN {X 0.086,Y -485.767,Z 679.524,A 0.000,B 0.000,C 90.000,E1 274.245} C_DIS
LIN {X -0.212,Y -486.701,Z 679.521,A 0.000,B 0.000,C 90.000,E1 273.784} C_DIS
LIN {X -0.049,Y -487.297,Z 679.518,A 0.000,B 0.000,C 90.000,E1 273.269} C_DIS
LIN {X 0.147,Y -487.601,Z 679.515,A 0.000,B 0.000,C 90.000,E1 272.751} C_DIS
LIN {X -0.165,Y -487.546,Z 679.513,A 0.000,B 0.000,C 90.000,E1 272.293} C_DIS
LIN {X 0.031,Y -487.231,Z 679.510,A 0.000,B 0.000,C 90.000,E1 271.776} C_DIS
LIN {X 0.209,Y -486.523,Z 679.507,A 0.000,B 0.000,C 90.000,E1 271.260} C_DIS
LIN {X -0.100,Y -485.408,Z 679.504,A 0.000,B 0.000,C 90.000,E1 270.802} C_DIS
LIN {X 0.074,Y -483.789,Z 679.502,A 0.000,B 0.000,C 90.000,E1 270.286} C_DIS
LIN {X 0.241,Y -481.632,Z 679.499,A 0.000,B 0.000,C 90.000,E1 269.771} C_DIS
LIN {X 0.078,Y -480.320,Z 679.497,A 0.000,B 0.000,C 90.000,E1 269.542} C_DIS
LIN {X 0.223,Y -477.035,Z 679.495,A 0.000,B 0.000,C 90.000,E1 269.026} C_DIS
LIN {X -0.126,Y -472.822,Z 679.492,A 0.000,B 0.000,C 90.000,E1 268.568} C_DIS
LIN {X 0.166,Y -470.365,Z 679.491,A 0.000,B 0.000,C 90.000,E1 268.282} C_DIS
LIN {X -0.160,Y -464.466,Z 679.488,A 0.000,B 0.000,C 90.000,E1 267.822} C_DIS
LIN {X -0.053,Y -461.485,Z 679.487,A 0.000,B 0.000,C 90.000,E1 267.593} C_DIS
LIN {X -0.008,Y -454.805,Z 679.484,A 0.000,B 0.000,C 90.000,E1 267.192} C_DIS
LIN {X 0.135,Y -447.689,Z 679.483,A 0.000,B 0.000,C 90.000,E1 266.849} C_DIS
LIN {X -0.107,Y -440.247,Z 679.481,A 0.000,B 0.000,C 90.000,E1 266.617} C_DIS
LIN {X 0.099,Y -432.158,Z 679.480,A 0.000,B 0.000,C 90.000,E1 266.388} C_DIS
LIN {X -0.016,Y -423.441,Z 679.479,A 0.000,B 0.000,C 90.000,E1 266.274} C_DIS
LIN {X 0.047,Y -416.134,Z 679.479,A 0.000,B 0.000,C 90.000,E1 266.216} C_DIS
LIN {X -0.005,Y -180.931,Z 679.479,A 0.000,B 0.000,C 90.000,E1 266.216} C_DIS
LIN {X 0.069,Y -180.763,Z 679.470,A 0.000,B 0.000,C 90.000,E1 264.666} C_DIS
LIN {X -0.073,Y -178.982,Z 679.444,A 0.000,B 0.000,C 90.000,E1 259.982} C_DIS
LIN {X -0.062,Y -177.954,Z 679.435,A 0.000,B 0.000,C 90.000,E1 258.285} C_DIS
LIN {X -0.042,Y -175.596,Z 679.411,A 0.000,B 0.000,C 90.000,E1 254.031} C_DIS
LIN {X -0.030,Y -172.320,Z 679.387,A 0.000,B 0.000,C 90.000,E1 249.752} C_DIS
LIN {X -0.051,Y -171.798,Z 679.383,A 0.000,B 0.000,C 90.000,E1 248.901} C_DIS
LIN {X -0.014,Y -169.470,Z 679.368,A 0.000,B 0.000,C 90.000,E1 246.305} C_DIS
LIN {X 0.042,Y -166.798,Z 679.349,A 0.000,B 0.000,C 90.000,E1 242.820} C_DIS
LIN {X 0.038,Y -162.778,Z 679.325,A 0.000,B 0.000,C 90.000,E1 238.456} C_DIS
LIN {X 0.013,Y -161.466,Z 679.315,A 0.000,B 0.000,C 90.000,E1 236.707} C_DIS
LIN {X 0.054,Y -157.462,Z 679.291,A 0.000,B 0.000,C 90.000,E1 232.271} C_DIS
LIN {X -0.014,Y -155.474,Z 679.276,A 0.000,B 0.000,C 90.000,E1 229.622} C_DIS
LIN {X -0.080,Y -151.785,Z 679.251,A 0.000,B 0.000,C 90.000,E1 225.162} C_DIS
LIN {X -0.066,Y -149.992,Z 679.236,A 0.000,B 0.000,C 90.000,E1 222.447} C_DIS
LIN {X -0.035,Y -146.823,Z 679.210,A 0.000,B 0.000,C 90.000,E1 217.890} C_DIS
LIN {X 0.071,Y -145.403,Z 679.195,A 0.000,B 0.000,C 90.000,E1 215.105} C_DIS
LIN {X -0.012,Y -142.835,Z 679.170,A 0.000,B 0.000,C 90.000,E1 210.541} C_DIS
LIN {X 0.044,Y -141.448,Z 679.149,A 0.000,B 0.000,C 90.000,E1 206.821} C_DIS
LIN {X -0.042,Y -139.371,Z 679.113,A 0.000,B 0.000,C 90.000,E1 200.355} C_DIS
LIN {X 0.033,Y -138.820,Z 679.097,A 0.000,B 0.000,C 90.000,E1 197.528} C_DIS
LIN {X -0.012,Y -138.352,Z 679.056,A 0.000,B 0.000,C 90.000,E1 190.074} C_DIS
LIN {X -0.038,Y -139.534,Z 679.004,A 0.000,B 0.000,C 90.000,E1 180.745} C_DIS
LIN {X 0.054,Y -141.220,Z 678.973,A 0.000,B 0.000,C 90.000,E1 175.122} C_DIS
LIN {X 0.014,Y -142.593,Z 678.958,A 0.000,B 0.000,C 90.000,E1 172.356} C_DIS
LIN {X -0.033,Y -144.895,Z 678.932,A 0.000,B 0.000,C 90.000,E1 167.757} C_DIS
LIN {X -0.079,Y -147.523,Z 678.911,A 0.000,B 0.000,C 90.000,E1 164.102} C_DIS
LIN {X -0.005,Y -150.120,Z 678.891,A 0.000,B 0.000,C 90.000,E1 160.423} C_DIS
LIN {X 0.006,Y -153.481,Z 678.871,A 0.000,B 0.000,C 90.000,E1 156.794} C_DIS
LIN {X 0.070,Y -157.845,Z 678.846,A 0.000,B 0.000,C 90.000,E1 152.281} C_DIS
LIN {X 0.026,Y -162.130,Z 678.826,A 0.000,B 0.000,C 90.000,E1 148.742} C_DIS
LIN {X 0.006,Y -166.333,Z 678.807,A 0.000,B 0.000,C 90.000,E1 145.229} C_DIS
LIN {X 0.012,Y -171.351,Z 678.787,A 0.000,B 0.000,C 90.000,E1 141.743} C_DIS
LIN {X -0.061,Y -176.254,Z 678.768,A 0.000,B 0.000,C 90.000,E1 138.324} C_DIS
LIN {X 0.058,Y -180.537,Z 678.754,A 0.000,B 0.000,C 90.000,E1 135.729} C_DIS
LIN {X 0.038,Y -185.939,Z 678.735,A 0.000,B 0.000,C 90.000,E1 132.366} C_DIS
LIN {X -0.036,Y -191.132,Z 678.720,A 0.000,B 0.000,C 90.000,E1 129.564} C_DIS
LIN {X -0.101,Y -289.294,Z 678.720,A 0.000,B 0.000,C 90.000,E1 129.564} C_DIS
LIN {X 0.077,Y -295.390,Z 678.718,A 0.000,B 0.000,C 90.000,E1 129.277} C_DIS
LIN {X 0.077,Y -298.083,Z 678.717,A 0.000,B 0.000,C 90.000,E1 129.036} C_DIS
LIN {X -0.075,Y -301.847,Z 678.714,A 0.000,B 0.000,C 90.000,E1 128.543} C_DIS
LIN {X 0.110,Y -303.520,Z 678.712,A 0.000,B 0.000,C 90.000,E1 128.177} C_DIS
LIN {X -0.131,Y -304.833,Z 678.710,A 0.000,B 0.000,C 90.000,E1 127.890} C_DIS
LIN {X -0.024,Y -315.443,Z 678.690,A 0.000,B 0.000,C 90.000,E1 124.278} C_DIS
LIN {X 0.023,Y -325.358,Z 678.674,A 0.000,B 0.000,C 90.000,E1 121.386} C_DIS
LIN {X -0.041,Y -336.589,Z 678.659,A 0.000,B 0.000,C 90.000,E1 118.565} C_DIS
LIN {X -0.097,Y -349.239,Z 678.643,A 0.000,B 0.000,C 90.000,E1 115.796} C_DIS
LIN {X -0.159,Y -361.765,Z 678.630,A 0.000,B 0.000,C 90.000,E1 113.387} C_DIS
LIN {X 0.140,Y -375.591,Z 678.617,A 0.000,B 0.000,C 90.000,E1 110.972} C_DIS
LIN {X 0.048,Y -390.815,Z 678.604,A 0.000,B 0.000,C 90.000,E1 108.671} C_DIS
LIN {X -0.168,Y -407.549,Z 678.591,A 0.000,B 0.000,C 90.000,E1 106.441} C_DIS
LIN {X -0.214,Y -425.915,Z 678.579,A 0.000,B 0.000,C 90.000,E1 104.245} C_DIS
LIN {X -0.102,Y -445.739,Z 678.567,A 0.000,B 0.000,C 90.000,E1 102.119} C_DIS
LIN {X -0.252,Y -466.187,Z 678.556,A 0.000,B 0.000,C 90.000,E1 100.197} C_DIS
LIN {X -0.204,Y -468.766,Z 678.555,A 0.000,B 0.000,C 90.000,E1 99.962} C_DIS
LIN {X -0.157,Y -470.972,Z 678.554,A 0.000,B 0.000,C 90.000,E1 99.726} C_DIS
LIN {X 0.084,Y -472.789,Z 678.552,A 0.000,B 0.000,C 90.000,E1 99.443} C_DIS
LIN {X -0.063,Y -474.155,Z 678.551,A 0.000,B 0.000,C 90.000,E1 99.208} C_DIS
LIN {X 0.125,Y -475.875,Z 678.548,A 0.000,B 0.000,C 90.000,E1 98.681} C_DIS
LIN {X 0.249,Y -476.520,Z 678.546,A 0.000,B 0.000,C 90.000,E1 98.163} C_DIS
LIN {X -0.087,Y -476.198,Z 678.543,A 0.000,B 0.000,C 90.000,E1 97.701} C_DIS
LIN {X 0.054,Y -474.861,Z 678.540,A 0.000,B 0.000,C 90.000,E1 97.182} C_DIS
LIN {X -0.083,Y -473.747,Z 678.539,A 0.000,B 0.000,C 90.000,E1 96.947} C_DIS
LIN {X 0.047,Y -470.533,Z 678.536,A 0.000,B 0.000,C 90.000,E1 96.429} C_DIS
LIN {X -0.091,Y -453.871,Z 678.522,A 0.000,B 0.000,C 90.000,E1 93.898} C_DIS
LIN {X 0.058,Y -436.240,Z 678.504,A 0.000,B 0.000,C 90.000,E1 90.745} C_DIS
LIN {X -0.026,Y -428.868,Z 678.497,A 0.000,B 0.000,C 90.000,E1 89.427} C_DIS
LIN {X 0.018,Y -418.000,Z 678.486,A 0.000,B 0.000,C 90.000,E1 87.535} C_DIS
LIN {X -0.133,Y -407.102,Z 678.476,A 0.000,B 0.000,C 90.000,E1 85.641} C_DIS
LIN {X 0.014,Y -393.120,Z 678.462,A 0.000,B 0.000,C 90.000,E1 83.109} C_DIS
LIN {X -0.058,Y -379.689,Z 678.448,A 0.000,B 0.000,C 90.000,E1 80.557} C_DIS
LIN {X -0.054,Y -366.718,Z 678.433,A 0.000,B 0.000,C 90.000,E1 77.937} C_DIS
LIN {X 0.157,Y -351.522,Z 678.415,A 0.000,B 0.000,C 90.000,E1 74.629} C_DIS
LIN {X -0.180,Y -339.678,Z 678.400,A 0.000,B 0.000,C 90.000,E1 71.945} C_DIS
LIN {X 0.166,Y -326.124,Z 678.380,A 0.000,B 0.000,C 90.000,E1 68.465} C_DIS
LIN {X 0.056,Y -314.892,Z 678.363,A 0.000,B 0.000,C 90.000,E1 65.305} C_DIS
LIN {X -0.040,Y -303.023,Z 678.341,A 0.000,B 0.000,C 90.000,E1 61.435} C_DIS
LIN {X 0.020,Y -294.079,Z 678.323,A 0.000,B 0.000,C 90.000,E1 58.122} C_DIS
LIN {X 0.014,Y -285.751,Z 678.304,A 0.000,B 0.000,C 90.000,E1 54.769} C_DIS
LIN {X -0.071,Y -279.132,Z 678.289,A 0.000,B 0.000,C 90.000,E1 52.065} C_DIS
LIN {X -0.008,Y -273.928,Z 678.278,A 0.000,B 0.000,C 90.000,E1 49.989} C_DIS
LIN {X -0.040,Y -270.325,Z 678.270,A 0.000,B 0.000,C 90.000,E1 48.609} C_DIS
LIN {X 0.014,Y -264.528,Z 678.258,A 0.000,B 0.000,C 90.000,E1 46.500} C_DIS
LIN {X 0.136,Y -258.469,Z 678.247,A 0.000,B 0.000,C 90.000,E1 44.352} C_DIS
LIN {X -0.030,Y -252.267,Z 678.235,A 0.000,B 0.000,C 90.000,E1 42.243} C_DIS
LIN {X -0.121,Y -245.913,Z 678.223,A 0.000,B 0.000,C 90.000,E1 40.092} C_DIS
LIN {X 0.017,Y -235.601,Z 678.202,A 0.000,B 0.000,C 90.000,E1 36.377} C_DIS
LIN {X 0.031,Y -227.907,Z 678.185,A 0.000,B 0.000,C 90.000,E1 33.372} C_DIS
LIN {X -0.013,Y -221.041,Z 678.169,A 0.000,B 0.000,C 90.000,E1 30.335} C_DIS
LIN {X -0.066,Y -214.992,Z 678.151,A 0.000,B 0.000,C 90.000,E1 27.257} C_DIS
LIN {X 0.108,Y -209.691,Z 678.134,A 0.000,B 0.000,C 90.000,E1 24.079} C_DIS
LIN {X 0.090,Y -204.274,Z 678.112,A 0.000,B 0.000,C 90.000,E1 20.120} C_DIS
LIN {X 0.012,Y -199.999,Z 678.090,A 0.000,B 0.000,C 90.000,E1 16.134} C_DIS
LIN {X -0.057,Y -196.301,Z 678.063,A 0.000,B 0.000,C 90.000,E1 11.299} C_DIS
LIN {X -0.016,Y -193.569,Z 678.026,A 0.000,B 0.000,C 90.000,E1 4.759} C_DIS
LIN {X -0.053,Y -195.121,Z 677.961,A 0.000,B 0.000,C 90.000,E1 352.996} C_DIS
LIN {X -0.053,Y -198.225,Z 677.934,A 0.000,B 0.000,C 90.000,E1 348.105} C_DIS
LIN {X 0.043,Y -201.952,Z 677.911,A 0.000,B 0.000,C 90.000,E1 344.031} C_DIS
LIN {X 0.086,Y -206.622,Z 677.889,A 0.000,B 0.000,C 90.000,E1 340.007} C_DIS
LIN {X 0.042,Y -212.095,Z 677.867,A 0.000,B 0.000,C 90.000,E1 336.049} C_DIS
LIN {X -0.059,Y -218.316,Z 677.845,A 0.000,B 0.000,C 90.000,E1 332.153} C_DIS
LIN {X -0.046,Y -225.258,Z 677.824,A 0.000,B 0.000,C 90.000,E1 328.280} C_DIS
LIN {X -0.111,Y -232.767,Z 677.803,A 0.000,B 0.000,C 90.000,E1 324.482} C_DIS
LIN {X -0.089,Y -240.969,Z 677.782,A 0.000,B 0.000,C 90.000,E1 320.723} C_DIS
LIN {X 0.110,Y -249.980,Z 677.761,A 0.000,B 0.000,C 90.000,E1 316.986} C_DIS
LIN {X 0.061,Y -260.180,Z 677.741,A 0.000,B 0.000,C 90.000,E1 313.380} C_DIS
LIN {X 0.138,Y -270.247,Z 677.723,A 0.000,B 0.000,C 90.000,E1 310.172} C_DIS
LIN {X -0.017,Y -281.554,Z 677.706,A 0.000,B 0.000,C 90.000,E1 307.076} C_DIS
LIN {X 0.092,Y -295.505,Z 677.687,A 0.000,B 0.000,C 90.000,E1 303.658} C_DIS
LIN {X -0.093,Y -310.755,Z 677.669,A 0.000,B 0.000,C 90.000,E1 300.384} C_DIS
LIN {X 0.120,Y -327.620,Z 677.651,A 0.000,B 0.000,C 90.000,E1 297.129} C_DIS
LIN {X 0.002,Y -343.768,Z 677.635,A 0.000,B 0.000,C 90.000,E1 294.335} C_DIS
LIN {X 0.106,Y -362.596,Z 677.618,A 0.000,B 0.000,C 90.000,E1 291.280} C_DIS
LIN {X 0.100,Y -374.774,Z 677.608,A 0.000,B 0.000,C 90.000,E1 289.504} C_DIS
LIN {X 0.028,Y -394.938,Z 677.594,A 0.000,B 0.000,C 90.000,E1 286.913} C_DIS
LIN {X -0.118,Y -408.992,Z 677.585,A 0.000,B 0.000,C 90.000,E1 285.245} C_DIS
LIN {X 0.156,Y -420.399,Z 677.577,A 0.000,B 0.000,C 90.000,E1 283.828} C_DIS
LIN {X 0.095,Y -431.352,Z 677.569,A 0.000,B 0.000,C 90.000,E1 282.479} C_DIS
LIN {X -0.002,Y -439.707,Z 677.563,A 0.000,B 0.000,C 90.000,E1 281.422} C_DIS
LIN {X 0.147,Y -449.528,Z 677.556,A 0.000,B 0.000,C 90.000,E1 280.084} C_DIS
LIN {X -0.151,Y -465.636,Z 677.545,A 0.000,B 0.000,C 90.000,E1 278.049} C_DIS
LIN {X 0.215,Y -471.349,Z 677.540,A 0.000,B 0.000,C 90.000,E1 277.239} C_DIS
LIN {X 0.170,Y -476.332,Z 677.536,A 0.000,B 0.000,C 90.000,E1 276.486} C_DIS
LIN {X -0.175,Y -479.115,Z 677.533,A 0.000,B 0.000,C 90.000,E1 276.024} C_DIS
LIN {X -0.075,Y -481.517,Z 677.531,A 0.000,B 0.000,C 90.000,E1 275.511} C_DIS
LIN {X -0.045,Y -484.321,Z 677.526,A 0.000,B 0.000,C 90.000,E1 274.759} C_DIS
LIN {X 0.093,Y -485.593,Z 677.524,A 0.000,B 0.000,C 90.000,E1 274.245} C_DIS
LIN {X -0.205,Y -486.573,Z 677.521,A 0.000,B 0.000,C 90.000,E1 273.784} C_DIS
LIN {X -0.044,Y -487.221,Z 677.518,A 0.000,B 0.000,C 90.000,E1 273.269} C_DIS
LIN {X 0.152,Y -487.503,Z 677.515,A 0.000,B 0.000,C 90.000,E1 272.751} C_DIS
LIN {X -0.160,Y -487.493,Z 677.513,A 0.000,B 0.000,C 90.000,E1 272.293} C_DIS
LIN {X 0.035,Y -487.132,Z 677.510,A 0.000,B 0.000,C 90.000,E1 271.776} C_DIS
LIN {X 0.212,Y -486.488,Z 677.507,A 0.000,B 0.000,C 90.000,E1 271.260} C_DIS
LIN {X -0.097,Y -485.374,Z 677.504,A 0.000,B 0.000,C 90.000,E1 270.802} C_DIS
LIN {X 0.077,Y -483.811,Z 677.502,A 0.000,B 0.000,C 90.000,E1 270.286} C_DIS
LIN {X -0.238,Y -481.638,Z 677.499,A 0.000,B 0.000,C 90.000,E1 269.828} C_DIS
LIN {X 0.079,Y -480.351,Z 677.497,A 0.000,B 0.000,C 90.000,E1 269.542} C_DIS
LIN {X 0.221,Y -477.050,Z 677.495,A 0.000,B 0.000,C 90.000,E1 269.026} C_DIS
LIN {X -0.129,Y -472.777,Z 677.492,A 0.000,B 0.000,C 90.000,E1 268.568} C_DIS
LIN {X 0.163,Y -470.352,Z 677.491,A 0.000,B 0.000,C 90.000,E1 268.282} C_DIS
LIN {X -0.194,Y -464.458,Z 677.488,A 0.000,B 0.000,C 90.000,E1 267.822} C_DIS
LIN {X -0.100,Y -461.422,Z 677.487,A 0.000,B 0.000,C 90.000,E1 267.593} C_DIS
LIN {X -0.066,Y -454.718,Z 677.484,A 0.000,B 0.000,C 90.000,E1 267.192} C_DIS
LIN {X 0.115,Y -447.613,Z 677.483,A 0.000,B 0.000,C 90.000,E1 266.846} C_DIS
LIN {X -0.118,Y -443.929,Z 677.482,A 0.000,B 0.000,C 90.000,E1 266.731} C_DIS
LIN {X -0.199,Y -435.706,Z 677.480,A 0.000,B 0.000,C 90.000,E1 266.502} C_DIS
LIN {X -0.162,Y -426.924,Z 677.479,A 0.000,B 0.000,C 90.000,E1 266.331} C_DIS
LIN {X 0.107,Y -418.907,Z 677.479,A 0.000,B 0.000,C 90.000,E1 266.216} C_DIS
LIN {X -0.014,Y -413.704,Z 677.479,A 0.000,B 0.000,C 90.000,E1 266.216} C_DIS
LIN {X -0.032,Y -180.929,Z 677.479,A 0.000,B 0.000,C 90.000,E1 266.216} C_DIS
LIN {X 0.041,Y -180.759,Z 677.470,A 0.000,B 0.000,C 90.000,E1 264.666} C_DIS
LIN {X 0.075,Y -178.979,Z 677.444,A 0.000,B 0.000,C 90.000,E1 259.926} C_DIS
LIN {X 0.085,Y -177.948,Z 677.435,A 0.000,B 0.000,C 90.000,E1 258.229} C_DIS
LIN {X -0.069,Y -175.589,Z 677.411,A 0.000,B 0.000,C 90.000,E1 254.031} C_DIS
LIN {X -0.056,Y -172.314,Z 677.387,A 0.000,B 0.000,C 90.000,E1 249.752} C_DIS
LIN {X -0.077,Y -171.792,Z 677.383,A 0.000,B 0.000,C 90.000,E1 248.901} C_DIS
LIN {X -0.039,Y -169.462,Z 677.368,A 0.000,B 0.000,C 90.000,E1 246.305} C_DIS
LIN {X 0.016,Y -166.791,Z 677.349,A 0.000,B 0.000,C 90.000,E1 242.820} C_DIS
LIN {X 0.012,Y -162.770,Z 677.325,A 0.000,B 0.000,C 90.000,E1 238.456} C_DIS
LIN {X -0.012,Y -161.460,Z 677.315,A 0.000,B 0.000,C 90.000,E1 236.707} C_DIS
LIN {X 0.029,Y -157.454,Z 677.290,A 0.000,B 0.000,C 90.000,E1 232.271} C_DIS
LIN {X -0.038,Y -155.465,Z 677.276,A 0.000,B 0.000,C 90.000,E1 229.622} C_DIS
LIN {X 0.003,Y -151.779,Z 677.251,A 0.000,B 0.000,C 90.000,E1 225.121} C_DIS
LIN {X 0.020,Y -149.985,Z 677.236,A 0.000,B 0.000,C 90.000,E1 222.405} C_DIS
LIN {X -0.059,Y -146.817,Z 677.210,A 0.000,B 0.000,C 90.000,E1 217.890} C_DIS
LIN {X 0.047,Y -145.396,Z 677.195,A 0.000,B 0.000,C 90.000,E1 215.105} C_DIS
LIN {X -0.035,Y -142.831,Z 677.170,A 0.000,B 0.000,C 90.000,E1 210.541} C_DIS
LIN {X 0.021,Y -141.444,Z 677.149,A 0.000,B 0.000,C 90.000,E1 206.821} C_DIS
LIN {X 0.065,Y -139.369,Z 677.113,A 0.000,B 0.000,C 90.000,E1 200.301} C_DIS
LIN {X 0.051,Y -138.817,Z 677.097,A 0.000,B 0.000,C 90.000,E1 197.511} C_DIS
LIN {X -0.034,Y -138.352,Z 677.056,A 0.000,B 0.000,C 90.000,E1 190.074} C_DIS
LIN {X -0.061,Y -139.536,Z 677.004,A 0.000,B 0.000,C 90.000,E1 180.745} C_DIS
LIN {X 0.032,Y -141.225,Z 676.973,A 0.000,B 0.000,C 90.000,E1 175.122} C_DIS
LIN {X -0.010,Y -142.596,Z 676.958,A 0.000,B 0.000,C 90.000,E1 172.356} C_DIS
LIN {X -0.056,Y -144.901,Z 676.932,A 0.000,B 0.000,C 90.000,E1 167.757} C_DIS
LIN {X 0.038,Y -147.529,Z 676.911,A 0.000,B 0.000,C 90.000,E1 164.047} C_DIS
LIN {X -0.030,Y -150.127,Z 676.891,A 0.000,B 0.000,C 90.000,E1 160.423} C_DIS
LIN {X -0.019,Y -153.491,Z 676.871,A 0.000,B 0.000,C 90.000,E1 156.794} C_DIS
LIN {X 0.045,Y -157.855,Z 676.846,A 0.000,B 0.000,C 90.000,E1 152.281} C_DIS
LIN {X 0.001,Y -162.141,Z 676.826,A 0.000,B 0.000,C 90.000,E1 148.742} C_DIS
LIN {X -0.021,Y -166.345,Z 676.807,A 0.000,B 0.000,C 90.000,E1 145.229} C_DIS
LIN {X -0.015,Y -171.362,Z 676.787,A 0.000,B 0.000,C 90.000,E1 141.743} C_DIS
LIN {X -0.087,Y -176.268,Z 676.768,A 0.000,B 0.000,C 90.000,E1 138.324} C_DIS
LIN {X 0.031,Y -180.552,Z 676.754,A 0.000,B 0.000,C 90.000,E1 135.729} C_DIS
LIN {X 0.010,Y -185.954,Z 676.735,A 0.000,B 0.000,C 90.000,E1 132.366} C_DIS
LIN {X 0.001,Y -191.115,Z 676.720,A 0.000,B 0.000,C 90.000,E1 129.564} C_DIS
LIN {X -0.047,Y -289.195,Z 676.720,A 0.000,B 0.000,C 90.000,E1 129.564} C_DIS
LIN {X 0.033,Y -290.773,Z 676.720,A 0.000,B 0.000,C 90.000,E1 129.519} C_DIS
LIN {X 0.034,Y -295.592,Z 676.718,A 0.000,B 0.000,C 90.000,E1 129.277} C_DIS
LIN {X 0.033,Y -298.209,Z 676.717,A 0.000,B 0.000,C 90.000,E1 129.036} C_DIS
LIN {X 0.004,Y -301.976,Z 676.714,A 0.000,B 0.000,C 90.000,E1 128.508} C_DIS
LIN {X 0.000,Y -303.610,Z 676.712,A 0.000,B 0.000,C 90.000,E1 128.177} C_DIS
LIN {X -0.054,Y -304.893,Z 676.710,A 0.000,B 0.000,C 90.000,E1 127.855} C_DIS
LIN {X 0.099,Y -316.529,Z 676.688,A 0.000,B 0.000,C 90.000,E1 123.913} C_DIS
LIN {X 0.004,Y -326.593,Z 676.673,A 0.000,B 0.000,C 90.000,E1 121.052} C_DIS
LIN {X -0.028,Y -337.987,Z 676.657,A 0.000,B 0.000,C 90.000,E1 118.231} C_DIS
LIN {X -0.045,Y -350.809,Z 676.641,A 0.000,B 0.000,C 90.000,E1 115.463} C_DIS
LIN {X 0.116,Y -363.502,Z 676.628,A 0.000,B 0.000,C 90.000,E1 113.025} C_DIS
LIN {X 0.124,Y -377.507,Z 676.615,A 0.000,B 0.000,C 90.000,E1 110.663} C_DIS
LIN {X 0.078,Y -392.925,Z 676.602,A 0.000,B 0.000,C 90.000,E1 108.362} C_DIS
LIN {X -0.091,Y -409.868,Z 676.590,A 0.000,B 0.000,C 90.000,E1 106.134} C_DIS
LIN {X -0.085,Y -428.460,Z 676.577,A 0.000,B 0.000,C 90.000,E1 103.939} C_DIS
LIN {X 0.094,Y -448.390,Z 676.566,A 0.000,B 0.000,C 90.000,E1 101.827} C_DIS
LIN {X 0.132,Y -468.907,Z 676.555,A 0.000,B 0.000,C 90.000,E1 99.905} C_DIS
LIN {X 0.182,Y -471.095,Z 676.554,A 0.000,B 0.000,C 90.000,E1 99.670} C_DIS
LIN {X -0.044,Y -472.904,Z 676.552,A 0.000,B 0.000,C 90.000,E1 99.443} C_DIS
LIN {X -0.194,Y -474.260,Z 676.551,A 0.000,B 0.000,C 90.000,E1 99.208} C_DIS
LIN {X -0.005,Y -475.965,Z 676.548,A 0.000,B 0.000,C 90.000,E1 98.681} C_DIS
LIN {X 0.119,Y -476.596,Z 676.545,A 0.000,B 0.000,C 90.000,E1 98.163} C_DIS
LIN {X -0.216,Y -476.259,Z 676.543,A 0.000,B 0.000,C 90.000,E1 97.701} C_DIS
LIN {X -0.074,Y -474.908,Z 676.540,A 0.000,B 0.000,C 90.000,E1 97.182} C_DIS
LIN {X -0.212,Y -473.784,Z 676.538,A 0.000,B 0.000,C 90.000,E1 96.947} C_DIS
LIN {X -0.080,Y -470.541,Z 676.536,A 0.000,B 0.000,C 90.000,E1 96.429} C_DIS
LIN {X -0.213,Y -453.884,Z 676.521,A 0.000,B 0.000,C 90.000,E1 93.898} C_DIS
LIN {X -0.058,Y -436.247,Z 676.504,A 0.000,B 0.000,C 90.000,E1 90.745} C_DIS
LIN {X -0.140,Y -428.879,Z 676.497,A 0.000,B 0.000,C 90.000,E1 89.427} C_DIS
LIN {X -0.093,Y -418.014,Z 676.486,A 0.000,B 0.000,C 90.000,E1 87.535} C_DIS
LIN {X 0.164,Y -407.113,Z 676.476,A 0.000,B 0.000,C 90.000,E1 85.584} C_DIS
LIN {X -0.109,Y -394.676,Z 676.463,A 0.000,B 0.000,C 90.000,E1 83.394} C_DIS
LIN {X 0.184,Y -381.213,Z 676.449,A 0.000,B 0.000,C 90.000,E1 80.792} C_DIS
LIN {X -0.138,Y -368.208,Z 676.435,A 0.000,B 0.000,C 90.000,E1 78.229} C_DIS
LIN {X 0.090,Y -354.300,Z 676.418,A 0.000,B 0.000,C 90.000,E1 75.227} C_DIS
LIN {X -0.173,Y -342.373,Z 676.403,A 0.000,B 0.000,C 90.000,E1 72.543} C_DIS
LIN {X -0.132,Y -329.827,Z 676.386,A 0.000,B 0.000,C 90.000,E1 69.444} C_DIS
LIN {X 0.123,Y -317.213,Z 676.366,A 0.000,B 0.000,C 90.000,E1 65.921} C_DIS
LIN {X -0.174,Y -305.096,Z 676.345,A 0.000,B 0.000,C 90.000,E1 62.103} C_DIS
LIN {X -0.052,Y -295.992,Z 676.327,A 0.000,B 0.000,C 90.000,E1 58.791} C_DIS
LIN {X -0.153,Y -287.596,Z 676.308,A 0.000,B 0.000,C 90.000,E1 55.468} C_DIS
LIN {X 0.039,Y -281.029,Z 676.293,A 0.000,B 0.000,C 90.000,E1 52.718} C_DIS
LIN {X -0.040,Y -275.924,Z 676.281,A 0.000,B 0.000,C 90.000,E1 50.678} C_DIS
LIN {X -0.069,Y -270.560,Z 676.270,A 0.000,B 0.000,C 90.000,E1 48.609} C_DIS
LIN {X -0.010,Y -264.773,Z 676.258,A 0.000,B 0.000,C 90.000,E1 46.500} C_DIS
LIN {X 0.118,Y -258.702,Z 676.247,A 0.000,B 0.000,C 90.000,E1 44.352} C_DIS
LIN {X -0.045,Y -252.469,Z 676.235,A 0.000,B 0.000,C 90.000,E1 42.243} C_DIS
LIN {X -0.132,Y -246.079,Z 676.223,A 0.000,B 0.000,C 90.000,E1 40.092} C_DIS
LIN {X 0.013,Y -235.776,Z 676.202,A 0.000,B 0.000,C 90.000,E1 36.377} C_DIS
LIN {X 0.030,Y -228.081,Z 676.185,A 0.000,B 0.000,C 90.000,E1 33.372} C_DIS
LIN {X -0.009,Y -221.212,Z 676.169,A 0.000,B 0.000,C 90.000,E1 30.335} C_DIS
LIN {X -0.057,Y -215.165,Z 676.151,A 0.000,B 0.000,C 90.000,E1 27.257} C_DIS
LIN {X -0.072,Y -209.855,Z 676.134,A 0.000,B 0.000,C 90.000,E1 24.131} C_DIS
LIN {X 0.107,Y -204.426,Z 676.112,A 0.000,B 0.000,C 90.000,E1 20.120} C_DIS
LIN {X 0.034,Y -200.140,Z 676.090,A 0.000,B 0.000,C 90.000,E1 16.134} C_DIS
LIN {X -0.031,Y -196.444,Z 676.063,A 0.000,B 0.000,C 90.000,E1 11.299} C_DIS
LIN {X 0.016,Y -193.681,Z 676.026,A 0.000,B 0.000,C 90.000,E1 4.759} C_DIS
LIN {X -0.048,Y -195.205,Z 675.961,A 0.000,B 0.000,C 90.000,E1 352.996} C_DIS
LIN {X -0.045,Y -198.294,Z 675.934,A 0.000,B 0.000,C 90.000,E1 348.105} C_DIS
LIN {X 0.052,Y -202.019,Z 675.911,A 0.000,B 0.000,C 90.000,E1 344.031} C_DIS
LIN {X -0.098,Y -206.684,Z 675.889,A 0.000,B 0.000,C 90.000,E1 340.061} C_DIS
LIN {X 0.056,Y -212.148,Z 675.867,A 0.000,B 0.000,C 90.000,E1 336.049} C_DIS
LIN {X -0.042,Y -218.373,Z 675.845,A 0.000,B 0.000,C 90.000,E1 332.153} C_DIS
LIN {X -0.028,Y -225.286,Z 675.824,A 0.000,B 0.000,C 90.000,E1 328.280} C_DIS
LIN {X -0.090,Y -232.812,Z 675.803,A 0.000,B 0.000,C 90.000,E1 324.482} C_DIS
LIN {X -0.067,Y -241.001,Z 675.782,A 0.000,B 0.000,C 90.000,E1 320.723} C_DIS
LIN {X -0.037,Y -249.989,Z 675.761,A 0.000,B 0.000,C 90.000,E1 317.025} C_DIS
LIN {X 0.085,Y -260.168,Z 675.741,A 0.000,B 0.000,C 90.000,E1 313.380} C_DIS
LIN {X -0.042,Y -270.228,Z 675.723,A 0.000,B 0.000,C 90.000,E1 310.216} C_DIS
LIN {X 0.009,Y -281.540,Z 675.706,A 0.000,B 0.000,C 90.000,E1 307.076} C_DIS
LIN {X -0.128,Y -295.466,Z 675.687,A 0.000,B 0.000,C 90.000,E1 303.706} C_DIS
LIN {X -0.066,Y -310.745,Z 675.669,A 0.000,B 0.000,C 90.000,E1 300.384} C_DIS
LIN {X 0.147,Y -327.586,Z 675.651,A 0.000,B 0.000,C 90.000,E1 297.129} C_DIS
LIN {X 0.031,Y -341.892,Z 675.637,A 0.000,B 0.000,C 90.000,E1 294.643} C_DIS
LIN {X 0.073,Y -360.557,Z 675.620,A 0.000,B 0.000,C 90.000,E1 291.589} C_DIS
LIN {X 0.030,Y -372.535,Z 675.610,A 0.000,B 0.000,C 90.000,E1 289.812} C_DIS
LIN {X -0.132,Y -390.186,Z 675.597,A 0.000,B 0.000,C 90.000,E1 287.511} C_DIS
LIN {X 0.212,Y -406.558,Z 675.586,A 0.000,B 0.000,C 90.000,E1 285.481} C_DIS
LIN {X 0.043,Y -418.031,Z 675.578,A 0.000,B 0.000,C 90.000,E1 284.120} C_DIS
LIN {X -0.051,Y -429.016,Z 675.571,A 0.000,B 0.000,C 90.000,E1 282.771} C_DIS
LIN {X -0.180,Y -437.508,Z 675.565,A 0.000,B 0.000,C 90.000,E1 281.715} C_DIS
LIN {X 0.222,Y -445.470,Z 675.559,A 0.000,B 0.000,C 90.000,E1 280.602} C_DIS
LIN {X -0.139,Y -465.501,Z 675.545,A 0.000,B 0.000,C 90.000,E1 278.049} C_DIS
LIN {X 0.226,Y -471.228,Z 675.540,A 0.000,B 0.000,C 90.000,E1 277.239} C_DIS
LIN {X -0.144,Y -474.636,Z 675.538,A 0.000,B 0.000,C 90.000,E1 276.777} C_DIS
LIN {X -0.022,Y -477.653,Z 675.535,A 0.000,B 0.000,C 90.000,E1 276.258} C_DIS
LIN {X -0.066,Y -481.376,Z 675.531,A 0.000,B 0.000,C 90.000,E1 275.511} C_DIS
LIN {X -0.037,Y -484.175,Z 675.526,A 0.000,B 0.000,C 90.000,E1 274.759} C_DIS
LIN {X 0.100,Y -485.488,Z 675.524,A 0.000,B 0.000,C 90.000,E1 274.245} C_DIS
LIN {X -0.199,Y -486.496,Z 675.521,A 0.000,B 0.000,C 90.000,E1 273.784} C_DIS
LIN {X -0.038,Y -487.119,Z 675.518,A 0.000,B 0.000,C 90.000,E1 273.269} C_DIS
LIN {X 0.157,Y -487.418,Z 675.515,A 0.000,B 0.000,C 90.000,E1 272.751} C_DIS
LIN {X -0.156,Y -487.404,Z 675.513,A 0.000,B 0.000,C 90.000,E1 272.293} C_DIS
LIN {X 0.038,Y -487.098,Z 675.510,A 0.000,B 0.000,C 90.000,E1 271.776} C_DIS
LIN {X 0.216,Y -486.455,Z 675.507,A 0.000,B 0.000,C 90.000,E1 271.260} C_DIS
LIN {X -0.094,Y -485.377,Z 675.504,A 0.000,B 0.000,C 90.000,E1 270.802} C_DIS
LIN {X 0.080,Y -483.819,Z 675.502,A 0.000,B 0.000,C 90.000,E1 270.286} C_DIS
LIN {X -0.235,Y -481.664,Z 675.499,A 0.000,B 0.000,C 90.000,E1 269.828} C_DIS
LIN {X 0.084,Y -480.362,Z 675.497,A 0.000,B 0.000,C 90.000,E1 269.542} C_DIS
LIN {X 0.230,Y -477.059,Z 675.495,A 0.000,B 0.000,C 90.000,E1 269.026} C_DIS
LIN {X 0.059,Y -475.089,Z 675.493,A 0.000,B 0.000,C 90.000,E1 268.797} C_DIS
LIN {X 0.172,Y -470.394,Z 675.491,A 0.000,B 0.000,C 90.000,E1 268.282} C_DIS
LIN {X -0.171,Y -464.533,Z 675.488,A 0.000,B 0.000,C 90.000,E1 267.822} C_DIS
LIN {X -0.073,Y -461.515,Z 675.487,A 0.000,B 0.000,C 90.000,E1 267.593} C_DIS
LIN {X 0.022,Y -458.077,Z 675.485,A 0.000,B 0.000,C 90.000,E1 267.364} C_DIS
LIN {X -0.112,Y -451.182,Z 675.483,A 0.000,B 0.000,C 90.000,E1 267.020} C_DIS
LIN {X -0.164,Y -443.861,Z 675.482,A 0.000,B 0.000,C 90.000,E1 266.731} C_DIS
LIN {X -0.200,Y -435.830,Z 675.480,A 0.000,B 0.000,C 90.000,E1 266.502} C_DIS
LIN {X -0.170,Y -427.087,Z 675.479,A 0.000,B 0.000,C 90.000,E1 266.331} C_DIS
LIN {X 0.093,Y -419.341,Z 675.479,A 0.000,B 0.000,C 90.000,E1 266.216} C_DIS
LIN {X -0.031,Y -414.897,Z 675.479,A 0.000,B 0.000,C 90.000,E1 266.216} C_DIS
LIN {X -0.040,Y -180.930,Z 675.479,A 0.000,B 0.000,C 90.000,E1 266.216} C_DIS
LIN {X 0.033,Y -180.758,Z 675.470,A 0.000,B 0.000,C 90.000,E1 264.666} C_DIS
LIN {X 0.067,Y -178.979,Z 675.444,A 0.000,B 0.000,C 90.000,E1 259.926} C_DIS
LIN {X 0.077,Y -177.946,Z 675.435,A 0.000,B 0.000,C 90.000,E1 258.229} C_DIS
LIN {X 0.091,Y -175.587,Z 675.411,A 0.000,B 0.000,C 90.000,E1 253.976} C_DIS
LIN {X -0.065,Y -172.312,Z 675.387,A 0.000,B 0.000,C 90.000,E1 249.752} C_DIS
LIN {X -0.086,Y -171.790,Z 675.383,A 0.000,B 0.000,C 90.000,E1 248.901} C_DIS
LIN {X -0.048,Y -169.459,Z 675.368,A 0.000,B 0.000,C 90.000,E1 246.305} C_DIS
LIN {X 0.008,Y -166.788,Z 675.349,A 0.000,B 0.000,C 90.000,E1 242.820} C_DIS
LIN {X 0.004,Y -162.769,Z 675.325,A 0.000,B 0.000,C 90.000,E1 238.456} C_DIS
LIN {X -0.021,Y -161.458,Z 675.315,A 0.000,B 0.000,C 90.000,E1 236.707} C_DIS
LIN {X 0.021,Y -157.452,Z 675.290,A 0.000,B 0.000,C 90.000,E1 232.271} C_DIS
LIN {X -0.046,Y -155.462,Z 675.276,A 0.000,B 0.000,C 90.000,E1 229.622} C_DIS
LIN {X -0.005,Y -151.777,Z 675.251,A 0.000,B 0.000,C 90.000,E1 225.121} C_DIS
LIN {X 0.012,Y -149.981,Z 675.236,A 0.000,B 0.000,C 90.000,E1 222.405} C_DIS
LIN {X -0.067,Y -146.816,Z 675.210,A 0.000,B 0.000,C 90.000,E1 217.890} C_DIS
LIN {X 0.039,Y -145.394,Z 675.195,A 0.000,B 0.000,C 90.000,E1 215.105} C_DIS
LIN {X -0.044,Y -142.829,Z 675.170,A 0.000,B 0.000,C 90.000,E1 210.541} C_DIS
LIN {X 0.013,Y -141.443,Z 675.149,A 0.000,B 0.000,C 90.000,E1 206.821} C_DIS
LIN {X 0.058,Y -139.368,Z 675.113,A 0.000,B 0.000,C 90.000,E1 200.301} C_DIS
LIN {X 0.043,Y -138.816,Z 675.097,A 0.000,B 0.000,C 90.000,E1 197.511} C_DIS
LIN {X -0.042,Y -138.352,Z 675.056,A 0.000,B 0.000,C 90.000,E1 190.074} C_DIS
LIN {X -0.069,Y -139.537,Z 675.004,A 0.000,B 0.000,C 90.000,E1 180.745} C_DIS
LIN {X 0.024,Y -141.225,Z 674.973,A 0.000,B 0.000,C 90.000,E1 175.122} C_DIS
LIN {X -0.017,Y -142.598,Z 674.958,A 0.000,B 0.000,C 90.000,E1 172.356} C_DIS
LIN {X -0.064,Y -144.903,Z 674.932,A 0.000,B 0.000,C 90.000,E1 167.757} C_DIS
LIN {X 0.031,Y -147.532,Z 674.911,A 0.000,B 0.000,C 90.000,E1 164.047} C_DIS
LIN {X -0.038,Y -150.129,Z 674.891,A 0.000,B 0.000,C 90.000,E1 160.423} C_DIS
LIN {X -0.027,Y -153.493,Z 674.871,A 0.000,B 0.000,C 90.000,E1 156.794} C_DIS
LIN {X 0.036,Y -157.858,Z 674.846,A 0.000,B 0.000,C 90.000,E1 152.281} C_DIS
LIN {X -0.008,Y -162.144,Z 674.826,A 0.000,B 0.000,C 90.000,E1 148.742} C_DIS
LIN {X -0.029,Y -166.349,Z 674.807,A 0.000,B 0.000,C 90.000,E1 145.229} C_DIS
LIN {X -0.023,Y -171.366,Z 674.787,A 0.000,B 0.000,C 90.000,E1 141.743} C_DIS
LIN {X -0.097,Y -176.273,Z 674.768,A 0.000,B 0.000,C 90.000,E1 138.324} C_DIS
LIN {X 0.022,Y -180.557,Z 674.754,A 0.000,B 0.000,C 90.000,E1 135.729} C_DIS
LIN {X 0.001,Y -185.959,Z 674.735,A 0.000,B 0.000,C 90.000,E1 132.366} C_DIS
LIN {X 0.038,Y -191.097,Z 674.720,A 0.000,B 0.000,C 90.000,E1 129.564} C_DIS
LIN {X 0.023,Y -288.853,Z 674.720,A 0.000,B 0.000,C 90.000,E1 129.564} C_DIS
LIN {X 0.020,Y -291.222,Z 674.720,A 0.000,B 0.000,C 90.000,E1 129.519} C_DIS
LIN {X 0.020,Y -295.727,Z 674.718,A 0.000,B 0.000,C 90.000,E1 129.277} C_DIS
LIN {X 0.018,Y -298.290,Z 674.717,A 0.000,B 0.000,C 90.000,E1 129.036} C_DIS
LIN {X 0.176,Y -302.057,Z 674.714,A 0.000,B 0.000,C 90.000,E1 128.463} C_DIS
LIN {X -0.063,Y -303.661,Z 674.712,A 0.000,B 0.000,C 90.000,E1 128.177} C_DIS
LIN {X 0.122,Y -304.922,Z 674.710,A 0.000,B 0.000,C 90.000,E1 127.810} C_DIS
LIN {X 0.034,Y -316.547,Z 674.688,A 0.000,B 0.000,C 90.000,E1 123.913} C_DIS
LIN {X -0.063,Y -326.615,Z 674.672,A 0.000,B 0.000,C 90.000,E1 121.052} C_DIS
LIN {X -0.096,Y -338.015,Z 674.657,A 0.000,B 0.000,C 90.000,E1 118.231} C_DIS
LIN {X -0.115,Y -350.843,Z 674.641,A 0.000,B 0.000,C 90.000,E1 115.463} C_DIS
LIN {X 0.044,Y -363.542,Z 674.628,A 0.000,B 0.000,C 90.000,E1 113.025} C_DIS
LIN {X 0.051,Y -377.553,Z 674.615,A 0.000,B 0.000,C 90.000,E1 110.663} C_DIS
LIN {X 0.003,Y -392.977,Z 674.602,A 0.000,B 0.000,C 90.000,E1 108.362} C_DIS
LIN {X 0.226,Y -409.928,Z 674.589,A 0.000,B 0.000,C 90.000,E1 106.079} C_DIS
LIN {X -0.164,Y -428.527,Z 674.577,A 0.000,B 0.000,C 90.000,E1 103.939} C_DIS
LIN {X 0.016,Y -448.461,Z 674.566,A 0.000,B 0.000,C 90.000,E1 101.827} C_DIS
LIN {X 0.056,Y -468.981,Z 674.555,A 0.000,B 0.000,C 90.000,E1 99.905} C_DIS
LIN {X 0.107,Y -471.167,Z 674.554,A 0.000,B 0.000,C 90.000,E1 99.670} C_DIS
LIN {X -0.119,Y -472.972,Z 674.552,A 0.000,B 0.000,C 90.000,E1 99.443} C_DIS
LIN {X 0.199,Y -474.328,Z 674.551,A 0.000,B 0.000,C 90.000,E1 99.151} C_DIS
LIN {X -0.080,Y -476.030,Z 674.548,A 0.000,B 0.000,C 90.000,E1 98.681} C_DIS
LIN {X 0.044,Y -476.659,Z 674.545,A 0.000,B 0.000,C 90.000,E1 98.163} C_DIS
LIN {X 0.182,Y -476.321,Z 674.543,A 0.000,B 0.000,C 90.000,E1 97.644} C_DIS
LIN {X -0.149,Y -474.967,Z 674.540,A 0.000,B 0.000,C 90.000,E1 97.182} C_DIS
LIN {X 0.185,Y -473.842,Z 674.538,A 0.000,B 0.000,C 90.000,E1 96.891} C_DIS
LIN {X -0.153,Y -470.592,Z 674.536,A 0.000,B 0.000,C 90.000,E1 96.429} C_DIS
LIN {X 0.171,Y -453.929,Z 674.521,A 0.000,B 0.000,C 90.000,E1 93.841} C_DIS
LIN {X -0.123,Y -436.289,Z 674.504,A 0.000,B 0.000,C 90.000,E1 90.745} C_DIS
LIN {X -0.204,Y -428.923,Z 674.497,A 0.000,B 0.000,C 90.000,E1 89.427} C_DIS
LIN {X 0.157,Y -419.628,Z 674.488,A 0.000,B 0.000,C 90.000,E1 87.764} C_DIS
LIN {X 0.107,Y -407.162,Z 674.476,A 0.000,B 0.000,C 90.000,E1 85.584} C_DIS
LIN {X -0.145,Y -393.233,Z 674.462,A 0.000,B 0.000,C 90.000,E1 83.109} C_DIS
LIN {X 0.165,Y -379.828,Z 674.447,A 0.000,B 0.000,C 90.000,E1 80.500} C_DIS
LIN {X 0.164,Y -366.904,Z 674.433,A 0.000,B 0.000,C 90.000,E1 77.881} C_DIS
LIN {X 0.029,Y -351.729,Z 674.415,A 0.000,B 0.000,C 90.000,E1 74.629} C_DIS
LIN {X 0.027,Y -338.670,Z 674.398,A 0.000,B 0.000,C 90.000,E1 71.583} C_DIS
LIN {X -0.013,Y -324.134,Z 674.377,A 0.000,B 0.000,C 90.000,E1 67.847} C_DIS
LIN {X -0.041,Y -313.183,Z 674.359,A 0.000,B 0.000,C 90.000,E1 64.665} C_DIS
LIN {X -0.113,Y -303.416,Z 674.341,A 0.000,B 0.000,C 90.000,E1 61.435} C_DIS
LIN {X -0.039,Y -294.501,Z 674.323,A 0.000,B 0.000,C 90.000,E1 58.122} C_DIS
LIN {X -0.030,Y -286.202,Z 674.304,A 0.000,B 0.000,C 90.000,E1 54.769} C_DIS
LIN {X 0.069,Y -279.605,Z 674.289,A 0.000,B 0.000,C 90.000,E1 52.029} C_DIS
LIN {X -0.031,Y -274.430,Z 674.278,A 0.000,B 0.000,C 90.000,E1 49.989} C_DIS
LIN {X -0.055,Y -270.818,Z 674.270,A 0.000,B 0.000,C 90.000,E1 48.609} C_DIS
LIN {X 0.008,Y -265.033,Z 674.258,A 0.000,B 0.000,C 90.000,E1 46.500} C_DIS
LIN {X 0.141,Y -258.962,Z 674.247,A 0.000,B 0.000,C 90.000,E1 44.352} C_DIS
LIN {X -0.018,Y -252.702,Z 674.235,A 0.000,B 0.000,C 90.000,E1 42.243} C_DIS
LIN {X -0.101,Y -246.269,Z 674.223,A 0.000,B 0.000,C 90.000,E1 40.092} C_DIS
LIN {X 0.047,Y -235.972,Z 674.202,A 0.000,B 0.000,C 90.000,E1 36.377} C_DIS
LIN {X 0.069,Y -228.280,Z 674.185,A 0.000,B 0.000,C 90.000,E1 33.372} C_DIS
LIN {X 0.033,Y -221.401,Z 674.169,A 0.000,B 0.000,C 90.000,E1 30.335} C_DIS
LIN {X -0.011,Y -215.357,Z 674.151,A 0.000,B 0.000,C 90.000,E1 27.257} C_DIS
LIN {X -0.023,Y -210.041,Z 674.134,A 0.000,B 0.000,C 90.000,E1 24.131} C_DIS
LIN {X -0.031,Y -204.593,Z 674.112,A 0.000,B 0.000,C 90.000,E1 20.174} C_DIS
LIN {X 0.036,Y -200.301,Z 674.090,A 0.000,B 0.000,C 90.000,E1 16.150} C_DIS
LIN {X 0.031,Y -196.593,Z 674.063,A 0.000,B 0.000,C 90.000,E1 11.299} C_DIS
LIN {X 0.084,Y -193.797,Z 674.027,A 0.000,B 0.000,C 90.000,E1 4.759} C_DIS
LIN {X -0.045,Y -195.293,Z 673.961,A 0.000,B 0.000,C 90.000,E1 352.996} C_DIS
LIN {X -0.039,Y -198.364,Z 673.934,A 0.000,B 0.000,C 90.000,E1 348.105} C_DIS
LIN {X 0.062,Y -202.083,Z 673.911,A 0.000,B 0.000,C 90.000,E1 344.031} C_DIS
LIN {X -0.085,Y -206.748,Z 673.889,A 0.000,B 0.000,C 90.000,E1 340.061} C_DIS
LIN {X 0.071,Y -212.203,Z 673.867,A 0.000,B 0.000,C 90.000,E1 336.049} C_DIS
LIN {X -0.026,Y -218.426,Z 673.845,A 0.000,B 0.000,C 90.000,E1 332.153} C_DIS
LIN {X -0.009,Y -225.331,Z 673.824,A 0.000,B 0.000,C 90.000,E1 328.280} C_DIS
LIN {X -0.070,Y -232.848,Z 673.803,A 0.000,B 0.000,C 90.000,E1 324.482} C_DIS
LIN {X -0.044,Y -241.014,Z 673.782,A 0.000,B 0.000,C 90.000,E1 320.723} C_DIS
LIN {X -0.013,Y -249.999,Z 673.761,A 0.000,B 0.000,C 90.000,E1 317.025} C_DIS
LIN {X -0.106,Y -259.107,Z 673.743,A 0.000,B 0.000,C 90.000,E1 313.785} C_DIS
LIN {X 0.109,Y -269.035,Z 673.725,A 0.000,B 0.000,C 90.000,E1 310.539} C_DIS
LIN {X -0.079,Y -280.191,Z 673.708,A 0.000,B 0.000,C 90.000,E1 307.443} C_DIS
LIN {X 0.150,Y -293.973,Z 673.689,A 0.000,B 0.000,C 90.000,E1 303.992} C_DIS
LIN {X -0.082,Y -309.136,Z 673.671,A 0.000,B 0.000,C 90.000,E1 300.718} C_DIS
LIN {X 0.078,Y -325.813,Z 673.653,A 0.000,B 0.000,C 90.000,E1 297.462} C_DIS
LIN {X 0.065,Y -340.016,Z 673.639,A 0.000,B 0.000,C 90.000,E1 294.951} C_DIS
LIN {X -0.001,Y -356.635,Z 673.623,A 0.000,B 0.000,C 90.000,E1 292.206} C_DIS
LIN {X 0.048,Y -372.423,Z 673.610,A 0.000,B 0.000,C 90.000,E1 289.812} C_DIS
LIN {X -0.116,Y -390.051,Z 673.597,A 0.000,B 0.000,C 90.000,E1 287.511} C_DIS
LIN {X 0.227,Y -406.428,Z 673.586,A 0.000,B 0.000,C 90.000,E1 285.481} C_DIS
LIN {X 0.056,Y -417.917,Z 673.578,A 0.000,B 0.000,C 90.000,E1 284.120} C_DIS
LIN {X -0.203,Y -426.730,Z 673.572,A 0.000,B 0.000,C 90.000,E1 283.063} C_DIS
LIN {X -0.170,Y -437.349,Z 673.565,A 0.000,B 0.000,C 90.000,E1 281.715} C_DIS
LIN {X 0.230,Y -445.313,Z 673.559,A 0.000,B 0.000,C 90.000,E1 280.602} C_DIS
LIN {X -0.135,Y -465.387,Z 673.545,A 0.000,B 0.000,C 90.000,E1 278.049} C_DIS
LIN {X 0.229,Y -471.125,Z 673.540,A 0.000,B 0.000,C 90.000,E1 277.239} C_DIS
LIN {X -0.141,Y -474.516,Z 673.538,A 0.000,B 0.000,C 90.000,E1 276.777} C_DIS
LIN {X -0.164,Y -478.848,Z 673.533,A 0.000,B 0.000,C 90.000,E1 276.024} C_DIS
LIN {X -0.066,Y -481.228,Z 673.531,A 0.000,B 0.000,C 90.000,E1 275.511} C_DIS
LIN {X -0.037,Y -484.050,Z 673.526,A 0.000,B 0.000,C 90.000,E1 274.759} C_DIS
LIN {X 0.099,Y -485.406,Z 673.524,A 0.000,B 0.000,C 90.000,E1 274.245} C_DIS
LIN {X -0.202,Y -486.416,Z 673.521,A 0.000,B 0.000,C 90.000,E1 273.784} C_DIS
LIN {X -0.041,Y -487.031,Z 673.518,A 0.000,B 0.000,C 90.000,E1 273.269} C_DIS
LIN {X 0.153,Y -487.364,Z 673.515,A 0.000,B 0.000,C 90.000,E1 272.751} C_DIS
LIN {X -0.160,Y -487.340,Z 673.513,A 0.000,B 0.000,C 90.000,E1 272.293} C_DIS
LIN {X 0.035,Y -487.063,Z 673.510,A 0.000,B 0.000,C 90.000,E1 271.776} C_DIS
LIN {X 0.211,Y -486.428,Z 673.507,A 0.000,B 0.000,C 90.000,E1 271.260} C_DIS
LIN {X -0.099,Y -485.372,Z 673.504,A 0.000,B 0.000,C 90.000,E1 270.802} C_DIS
LIN {X 0.075,Y -483.835,Z 673.502,A 0.000,B 0.000,C 90.000,E1 270.286} C_DIS
LIN {X -0.240,Y -481.674,Z 673.499,A 0.000,B 0.000,C 90.000,E1 269.828} C_DIS
LIN {X -0.082,Y -478.805,Z 673.496,A 0.000,B 0.000,C 90.000,E1 269.312} C_DIS
LIN {X 0.054,Y -475.102,Z 673.493,A 0.000,B 0.000,C 90.000,E1 268.797} C_DIS
LIN {X 0.168,Y -470.435,Z 673.491,A 0.000,B 0.000,C 90.000,E1 268.282} C_DIS
LIN {X -0.149,Y -464.624,Z 673.488,A 0.000,B 0.000,C 90.000,E1 267.822} C_DIS
LIN {X -0.053,Y -461.634,Z 673.487,A 0.000,B 0.000,C 90.000,E1 267.593} C_DIS
LIN {X -0.027,Y -454.981,Z 673.484,A 0.000,B 0.000,C 90.000,E1 267.192} C_DIS
LIN {X 0.114,Y -447.931,Z 673.483,A 0.000,B 0.000,C 90.000,E1 266.846} C_DIS
LIN {X -0.158,Y -440.331,Z 673.481,A 0.000,B 0.000,C 90.000,E1 266.617} C_DIS
LIN {X 0.046,Y -432.217,Z 673.480,A 0.000,B 0.000,C 90.000,E1 266.388} C_DIS
LIN {X -0.080,Y -423.840,Z 673.479,A 0.000,B 0.000,C 90.000,E1 266.274} C_DIS
LIN {X -0.039,Y -416.890,Z 673.479,A 0.000,B 0.000,C 90.000,E1 266.216} C_DIS
LIN {X -0.044,Y -180.929,Z 673.479,A 0.000,B 0.000,C 90.000,E1 266.216} C_DIS
LIN {X 0.028,Y -180.757,Z 673.470,A 0.000,B 0.000,C 90.000,E1 264.666} C_DIS
LIN {X 0.062,Y -178.978,Z 673.444,A 0.000,B 0.000,C 90.000,E1 259.926} C_DIS
LIN {X 0.072,Y -177.945,Z 673.435,A 0.000,B 0.000,C 90.000,E1 258.229} C_DIS
LIN {X 0.086,Y -175.585,Z 673.411,A 0.000,B 0.000,C 90.000,E1 253.976} C_DIS
LIN {X -0.069,Y -172.312,Z 673.387,A 0.000,B 0.000,C 90.000,E1 249.752} C_DIS
LIN {X -0.091,Y -171.790,Z 673.383,A 0.000,B 0.000,C 90.000,E1 248.901} C_DIS
LIN {X -0.053,Y -169.458,Z 673.368,A 0.000,B 0.000,C 90.000,E1 246.305} C_DIS
LIN {X 0.003,Y -166.788,Z 673.349,A 0.000,B 0.000,C 90.000,E1 242.820} C_DIS
LIN {X -0.001,Y -162.768,Z 673.325,A 0.000,B 0.000,C 90.000,E1 238.456} C_DIS
LIN {X -0.025,Y -161.457,Z 673.315,A 0.000,B 0.000,C 90.000,E1 236.707} C_DIS
LIN {X 0.016,Y -157.450,Z 673.290,A 0.000,B 0.000,C 90.000,E1 232.271} C_DIS
LIN {X -0.051,Y -155.461,Z 673.276,A 0.000,B 0.000,C 90.000,E1 229.622} C_DIS
LIN {X -0.009,Y -151.775,Z 673.251,A 0.000,B 0.000,C 90.000,E1 225.121} C_DIS
LIN {X 0.008,Y -149.980,Z 673.236,A 0.000,B 0.000,C 90.000,E1 222.405} C_DIS
LIN {X -0.071,Y -146.815,Z 673.210,A 0.000,B 0.000,C 90.000,E1 217.890} C_DIS
LIN {X 0.034,Y -145.394,Z 673.195,A 0.000,B 0.000,C 90.000,E1 215.105} C_DIS
LIN {X -0.048,Y -142.829,Z 673.170,A 0.000,B 0.000,C 90.000,E1 210.541} C_DIS
LIN {X 0.009,Y -141.442,Z 673.149,A 0.000,B 0.000,C 90.000,E1 206.821} C_DIS
LIN {X 0.053,Y -139.369,Z 673.113,A 0.000,B 0.000,C 90.000,E1 200.301} C_DIS
LIN {X 0.039,Y -138.816,Z 673.097,A 0.000,B 0.000,C 90.000,E1 197.511} C_DIS
LIN {X -0.046,Y -138.352,Z 673.056,A 0.000,B 0.000,C 90.000,E1 190.074} C_DIS
LIN {X 0.067,Y -139.537,Z 673.004,A 0.000,B 0.000,C 90.000,E1 180.688} C_DIS
LIN {X 0.020,Y -141.227,Z 672.973,A 0.000,B 0.000,C 90.000,E1 175.122} C_DIS
LIN {X -0.021,Y -142.599,Z 672.957,A 0.000,B 0.000,C 90.000,E1 172.356} C_DIS
LIN {X 0.073,Y -144.904,Z 672.932,A 0.000,B 0.000,C 90.000,E1 167.701} C_DIS
LIN {X 0.026,Y -147.533,Z 672.911,A 0.000,B 0.000,C 90.000,E1 164.047} C_DIS
LIN {X -0.042,Y -150.131,Z 672.891,A 0.000,B 0.000,C 90.000,E1 160.423} C_DIS
LIN {X -0.031,Y -153.495,Z 672.871,A 0.000,B 0.000,C 90.000,E1 156.794} C_DIS
LIN {X 0.032,Y -157.860,Z 672.846,A 0.000,B 0.000,C 90.000,E1 152.281} C_DIS
LIN {X -0.013,Y -162.145,Z 672.826,A 0.000,B 0.000,C 90.000,E1 148.742} C_DIS
LIN {X -0.034,Y -166.351,Z 672.807,A 0.000,B 0.000,C 90.000,E1 145.229} C_DIS
LIN {X -0.028,Y -171.368,Z 672.787,A 0.000,B 0.000,C 90.000,E1 141.743} C_DIS
LIN {X -0.101,Y -176.275,Z 672.768,A 0.000,B 0.000,C 90.000,E1 138.324} C_DIS
LIN {X 0.017,Y -180.559,Z 672.754,A 0.000,B 0.000,C 90.000,E1 135.729} C_DIS
LIN {X -0.004,Y -185.961,Z 672.735,A 0.000,B 0.000,C 90.000,E1 132.366} C_DIS
LIN {X 0.057,Y -191.088,Z 672.720,A 0.000,B 0.000,C 90.000,E1 129.564} C_DIS
LIN {X 0.050,Y -289.036,Z 672.720,A 0.000,B 0.000,C 90.000,E1 129.564} C_DIS
LIN {X 0.012,Y -291.461,Z 672.720,A 0.000,B 0.000,C 90.000,E1 129.519} C_DIS
LIN {X 0.012,Y -295.799,Z 672.718,A 0.000,B 0.000,C 90.000,E1 129.277} C_DIS
LIN {X 0.011,Y -298.329,Z 672.717,A 0.000,B 0.000,C 90.000,E1 129.036} C_DIS
LIN {X 0.138,Y -302.097,Z 672.714,A 0.000,B 0.000,C 90.000,E1 128.463} C_DIS
LIN {X -0.103,Y -303.683,Z 672.712,A 0.000,B 0.000,C 90.000,E1 128.177} C_DIS
LIN {X 0.084,Y -304.931,Z 672.710,A 0.000,B 0.000,C 90.000,E1 127.810} C_DIS
LIN {X -0.006,Y -316.549,Z 672.688,A 0.000,B 0.000,C 90.000,E1 123.913} C_DIS
LIN {X -0.103,Y -326.620,Z 672.672,A 0.000,B 0.000,C 90.000,E1 121.052} C_DIS
LIN {X -0.139,Y -338.024,Z 672.657,A 0.000,B 0.000,C 90.000,E1 118.231} C_DIS
LIN {X -0.159,Y -350.856,Z 672.641,A 0.000,B 0.000,C 90.000,E1 115.463} C_DIS
LIN {X 0.000,Y -363.557,Z 672.628,A 0.000,B 0.000,C 90.000,E1 113.025} C_DIS
LIN {X 0.004,Y -377.572,Z 672.615,A 0.000,B 0.000,C 90.000,E1 110.663} C_DIS
LIN {X -0.044,Y -393.001,Z 672.602,A 0.000,B 0.000,C 90.000,E1 108.362} C_DIS
LIN {X 0.177,Y -409.956,Z 672.589,A 0.000,B 0.000,C 90.000,E1 106.079} C_DIS
LIN {X 0.201,Y -428.560,Z 672.577,A 0.000,B 0.000,C 90.000,E1 103.883} C_DIS
LIN {X -0.033,Y -448.496,Z 672.566,A 0.000,B 0.000,C 90.000,E1 101.827} C_DIS
LIN {X 0.008,Y -469.019,Z 672.555,A 0.000,B 0.000,C 90.000,E1 99.905} C_DIS
LIN {X 0.059,Y -471.211,Z 672.554,A 0.000,B 0.000,C 90.000,E1 99.670} C_DIS
LIN {X -0.091,Y -473.023,Z 672.552,A 0.000,B 0.000,C 90.000,E1 99.434} C_DIS
LIN {X 0.151,Y -474.383,Z 672.551,A 0.000,B 0.000,C 90.000,E1 99.151} C_DIS
LIN {X -0.128,Y -476.093,Z 672.548,A 0.000,B 0.000,C 90.000,E1 98.681} C_DIS
LIN {X -0.003,Y -476.728,Z 672.545,A 0.000,B 0.000,C 90.000,E1 98.163} C_DIS
LIN {X 0.133,Y -476.396,Z 672.543,A 0.000,B 0.000,C 90.000,E1 97.644} C_DIS
LIN {X -0.196,Y -475.049,Z 672.540,A 0.000,B 0.000,C 90.000,E1 97.182} C_DIS
LIN {X 0.138,Y -473.928,Z 672.538,A 0.000,B 0.000,C 90.000,E1 96.891} C_DIS
LIN {X -0.055,Y -472.430,Z 672.537,A 0.000,B 0.000,C 90.000,E1 96.663} C_DIS
LIN {X -0.126,Y -455.586,Z 672.523,A 0.000,B 0.000,C 90.000,E1 94.131} C_DIS
LIN {X 0.010,Y -442.059,Z 672.510,A 0.000,B 0.000,C 90.000,E1 91.776} C_DIS
LIN {X 0.165,Y -433.458,Z 672.501,A 0.000,B 0.000,C 90.000,E1 90.172} C_DIS
LIN {X 0.038,Y -425.911,Z 672.494,A 0.000,B 0.000,C 90.000,E1 88.854} C_DIS
LIN {X 0.016,Y -415.002,Z 672.483,A 0.000,B 0.000,C 90.000,E1 86.963} C_DIS
LIN {X -0.170,Y -404.115,Z 672.472,A 0.000,B 0.000,C 90.000,E1 85.065} C_DIS
LIN {X -0.050,Y -390.316,Z 672.458,A 0.000,B 0.000,C 90.000,E1 82.527} C_DIS
LIN {X 0.122,Y -377.011,Z 672.444,A 0.000,B 0.000,C 90.000,E1 79.926} C_DIS
LIN {X 0.131,Y -365.634,Z 672.431,A 0.000,B 0.000,C 90.000,E1 77.589} C_DIS
LIN {X -0.053,Y -350.555,Z 672.413,A 0.000,B 0.000,C 90.000,E1 74.338} C_DIS
LIN {X 0.013,Y -337.589,Z 672.396,A 0.000,B 0.000,C 90.000,E1 71.275} C_DIS
LIN {X -0.061,Y -323.192,Z 672.375,A 0.000,B 0.000,C 90.000,E1 67.539} C_DIS
LIN {X -0.057,Y -311.375,Z 672.356,A 0.000,B 0.000,C 90.000,E1 64.024} C_DIS
LIN {X -0.183,Y -301.779,Z 672.338,A 0.000,B 0.000,C 90.000,E1 60.795} C_DIS
LIN {X -0.012,Y -293.030,Z 672.319,A 0.000,B 0.000,C 90.000,E1 57.454} C_DIS
LIN {X -0.008,Y -286.444,Z 672.304,A 0.000,B 0.000,C 90.000,E1 54.769} C_DIS
LIN {X -0.075,Y -279.859,Z 672.289,A 0.000,B 0.000,C 90.000,E1 52.065} C_DIS
LIN {X 0.001,Y -274.692,Z 672.278,A 0.000,B 0.000,C 90.000,E1 49.989} C_DIS
LIN {X -0.047,Y -269.190,Z 672.266,A 0.000,B 0.000,C 90.000,E1 47.919} C_DIS
LIN {X -0.017,Y -263.312,Z 672.254,A 0.000,B 0.000,C 90.000,E1 45.810} C_DIS
LIN {X -0.103,Y -257.153,Z 672.243,A 0.000,B 0.000,C 90.000,E1 43.704} C_DIS
LIN {X 0.063,Y -250.810,Z 672.231,A 0.000,B 0.000,C 90.000,E1 41.515} C_DIS
LIN {X -0.026,Y -242.255,Z 672.215,A 0.000,B 0.000,C 90.000,E1 38.624} C_DIS
LIN {X 0.044,Y -232.261,Z 672.194,A 0.000,B 0.000,C 90.000,E1 34.898} C_DIS
LIN {X 0.038,Y -224.926,Z 672.177,A 0.000,B 0.000,C 90.000,E1 31.878} C_DIS
LIN {X -0.002,Y -218.467,Z 672.160,A 0.000,B 0.000,C 90.000,E1 28.821} C_DIS
LIN {X -0.029,Y -212.784,Z 672.143,A 0.000,B 0.000,C 90.000,E1 25.720} C_DIS
LIN {X -0.083,Y -207.898,Z 672.125,A 0.000,B 0.000,C 90.000,E1 22.589} C_DIS
LIN {X -0.033,Y -202.942,Z 672.103,A 0.000,B 0.000,C 90.000,E1 18.598} C_DIS
LIN {X -0.077,Y -199.077,Z 672.081,A 0.000,B 0.000,C 90.000,E1 14.592} C_DIS
LIN {X -0.070,Y -195.791,Z 672.054,A 0.000,B 0.000,C 90.000,E1 9.726} C_DIS
LIN {X 0.012,Y -193.527,Z 672.013,A 0.000,B 0.000,C 90.000,E1 2.350} C_DIS
LIN {X -0.040,Y -195.380,Z 671.961,A 0.000,B 0.000,C 90.000,E1 352.996} C_DIS
LIN {X -0.032,Y -198.437,Z 671.934,A 0.000,B 0.000,C 90.000,E1 348.105} C_DIS
LIN {X 0.016,Y -202.146,Z 671.911,A 0.000,B 0.000,C 90.000,E1 344.047} C_DIS
LIN {X -0.073,Y -206.813,Z 671.889,A 0.000,B 0.000,C 90.000,E1 340.061} C_DIS
LIN {X 0.085,Y -212.259,Z 671.867,A 0.000,B 0.000,C 90.000,E1 336.049} C_DIS
LIN {X -0.010,Y -218.482,Z 671.845,A 0.000,B 0.000,C 90.000,E1 332.153} C_DIS
LIN {X 0.010,Y -225.377,Z 671.824,A 0.000,B 0.000,C 90.000,E1 328.280} C_DIS
LIN {X -0.049,Y -232.880,Z 671.803,A 0.000,B 0.000,C 90.000,E1 324.482} C_DIS
LIN {X -0.021,Y -241.038,Z 671.782,A 0.000,B 0.000,C 90.000,E1 320.723} C_DIS
LIN {X 0.012,Y -250.009,Z 671.761,A 0.000,B 0.000,C 90.000,E1 317.025} C_DIS
LIN {X -0.080,Y -259.084,Z 671.743,A 0.000,B 0.000,C 90.000,E1 313.785} C_DIS
LIN {X 0.135,Y -269.012,Z 671.725,A 0.000,B 0.000,C 90.000,E1 310.539} C_DIS
LIN {X -0.053,Y -280.159,Z 671.708,A 0.000,B 0.000,C 90.000,E1 307.443} C_DIS
LIN {X -0.068,Y -293.920,Z 671.689,A 0.000,B 0.000,C 90.000,E1 304.040} C_DIS
LIN {X -0.056,Y -309.113,Z 671.671,A 0.000,B 0.000,C 90.000,E1 300.718} C_DIS
LIN {X 0.106,Y -325.772,Z 671.653,A 0.000,B 0.000,C 90.000,E1 297.462} C_DIS
LIN {X 0.092,Y -339.958,Z 671.639,A 0.000,B 0.000,C 90.000,E1 294.951} C_DIS
LIN {X 0.026,Y -356.546,Z 671.623,A 0.000,B 0.000,C 90.000,E1 292.206} C_DIS
LIN {X 0.073,Y -372.304,Z 671.610,A 0.000,B 0.000,C 90.000,E1 289.812} C_DIS
LIN {X -0.093,Y -389.911,Z 671.597,A 0.000,B 0.000,C 90.000,E1 287.511} C_DIS
LIN {X -0.144,Y -406.286,Z 671.586,A 0.000,B 0.000,C 90.000,E1 285.536} C_DIS
LIN {X 0.075,Y -417.791,Z 671.578,A 0.000,B 0.000,C 90.000,E1 284.120} C_DIS
LIN {X -0.184,Y -426.605,Z 671.572,A 0.000,B 0.000,C 90.000,E1 283.063} C_DIS
LIN {X 0.081,Y -435.116,Z 671.566,A 0.000,B 0.000,C 90.000,E1 281.951} C_DIS
LIN {X 0.024,Y -443.222,Z 671.561,A 0.000,B 0.000,C 90.000,E1 280.894} C_DIS
LIN {X -0.123,Y -465.294,Z 671.545,A 0.000,B 0.000,C 90.000,E1 278.049} C_DIS
LIN {X -0.227,Y -471.034,Z 671.540,A 0.000,B 0.000,C 90.000,E1 277.296} C_DIS
LIN {X -0.130,Y -474.410,Z 671.538,A 0.000,B 0.000,C 90.000,E1 276.777} C_DIS
LIN {X -0.011,Y -477.393,Z 671.535,A 0.000,B 0.000,C 90.000,E1 276.258} C_DIS
LIN {X -0.056,Y -481.100,Z 671.531,A 0.000,B 0.000,C 90.000,E1 275.511} C_DIS
LIN {X -0.196,Y -482.160,Z 671.529,A 0.000,B 0.000,C 90.000,E1 275.277} C_DIS
LIN {X -0.029,Y -483.941,Z 671.526,A 0.000,B 0.000,C 90.000,E1 274.759} C_DIS
LIN {X 0.106,Y -485.336,Z 671.524,A 0.000,B 0.000,C 90.000,E1 274.245} C_DIS
LIN {X -0.195,Y -486.329,Z 671.521,A 0.000,B 0.000,C 90.000,E1 273.784} C_DIS
LIN {X -0.035,Y -486.988,Z 671.518,A 0.000,B 0.000,C 90.000,E1 273.269} C_DIS
LIN {X 0.160,Y -487.328,Z 671.515,A 0.000,B 0.000,C 90.000,E1 272.751} C_DIS
LIN {X -0.154,Y -487.314,Z 671.513,A 0.000,B 0.000,C 90.000,E1 272.293} C_DIS
LIN {X 0.040,Y -487.037,Z 671.510,A 0.000,B 0.000,C 90.000,E1 271.776} C_DIS
LIN {X 0.217,Y -486.404,Z 671.507,A 0.000,B 0.000,C 90.000,E1 271.260} C_DIS
LIN {X -0.094,Y -485.369,Z 671.504,A 0.000,B 0.000,C 90.000,E1 270.802} C_DIS
LIN {X 0.080,Y -483.833,Z 671.502,A 0.000,B 0.000,C 90.000,E1 270.286} C_DIS
LIN {X -0.235,Y -481.702,Z 671.499,A 0.000,B 0.000,C 90.000,E1 269.828} C_DIS
LIN {X -0.077,Y -478.849,Z 671.496,A 0.000,B 0.000,C 90.000,E1 269.312} C_DIS
LIN {X 0.059,Y -475.185,Z 671.493,A 0.000,B 0.000,C 90.000,E1 268.797} C_DIS
LIN {X -0.120,Y -472.993,Z 671.492,A 0.000,B 0.000,C 90.000,E1 268.568} C_DIS
LIN {X 0.048,Y -467.810,Z 671.489,A 0.000,B 0.000,C 90.000,E1 268.051} C_DIS
LIN {X 0.019,Y -461.809,Z 671.487,A 0.000,B 0.000,C 90.000,E1 267.593} C_DIS
LIN {X 0.043,Y -455.238,Z 671.484,A 0.000,B 0.000,C 90.000,E1 267.192} C_DIS
LIN {X 0.148,Y -448.200,Z 671.483,A 0.000,B 0.000,C 90.000,E1 266.849} C_DIS
LIN {X -0.113,Y -440.735,Z 671.481,A 0.000,B 0.000,C 90.000,E1 266.617} C_DIS
LIN {X 0.084,Y -432.604,Z 671.480,A 0.000,B 0.000,C 90.000,E1 266.388} C_DIS
LIN {X -0.036,Y -424.613,Z 671.479,A 0.000,B 0.000,C 90.000,E1 266.274} C_DIS
LIN {X -0.083,Y -415.664,Z 671.479,A 0.000,B 0.000,C 90.000,E1 266.216} C_DIS
LIN {X -0.065,Y -180.930,Z 671.479,A 0.000,B 0.000,C 90.000,E1 266.216} C_DIS
LIN {X 0.007,Y -180.754,Z 671.470,A 0.000,B 0.000,C 90.000,E1 264.666} C_DIS
LIN {X 0.041,Y -178.976,Z 671.444,A 0.000,B 0.000,C 90.000,E1 259.926} C_DIS
LIN {X 0.051,Y -177.941,Z 671.435,A 0.000,B 0.000,C 90.000,E1 258.229} C_DIS
LIN {X 0.066,Y -175.581,Z 671.411,A 0.000,B 0.000,C 90.000,E1 253.976} C_DIS
LIN {X 0.073,Y -172.307,Z 671.387,A 0.000,B 0.000,C 90.000,E1 249.699} C_DIS
LIN {X 0.050,Y -171.786,Z 671.383,A 0.000,B 0.000,C 90.000,E1 248.847} C_DIS
LIN {X -0.073,Y -169.452,Z 671.368,A 0.000,B 0.000,C 90.000,E1 246.305} C_DIS
LIN {X -0.017,Y -166.782,Z 671.349,A 0.000,B 0.000,C 90.000,E1 242.820} C_DIS
LIN {X -0.020,Y -162.762,Z 671.325,A 0.000,B 0.000,C 90.000,E1 238.456} C_DIS
LIN {X -0.045,Y -161.452,Z 671.315,A 0.000,B 0.000,C 90.000,E1 236.707} C_DIS
LIN {X -0.003,Y -157.446,Z 671.290,A 0.000,B 0.000,C 90.000,E1 232.271} C_DIS
LIN {X -0.070,Y -155.455,Z 671.276,A 0.000,B 0.000,C 90.000,E1 229.622} C_DIS
LIN {X 0.079,Y -151.771,Z 671.251,A 0.000,B 0.000,C 90.000,E1 225.081} C_DIS
LIN {X -0.011,Y -149.974,Z 671.236,A 0.000,B 0.000,C 90.000,E1 222.405} C_DIS
LIN {X 0.000,Y -146.811,Z 671.210,A 0.000,B 0.000,C 90.000,E1 217.855} C_DIS
LIN {X 0.017,Y -145.389,Z 671.195,A 0.000,B 0.000,C 90.000,E1 215.105} C_DIS
LIN {X -0.066,Y -142.825,Z 671.170,A 0.000,B 0.000,C 90.000,E1 210.541} C_DIS
LIN {X -0.009,Y -141.438,Z 671.149,A 0.000,B 0.000,C 90.000,E1 206.821} C_DIS
LIN {X 0.036,Y -139.368,Z 671.113,A 0.000,B 0.000,C 90.000,E1 200.301} C_DIS
LIN {X 0.022,Y -138.814,Z 671.097,A 0.000,B 0.000,C 90.000,E1 197.511} C_DIS
LIN {X 0.073,Y -138.351,Z 671.056,A 0.000,B 0.000,C 90.000,E1 190.018} C_DIS
LIN {X 0.049,Y -139.538,Z 671.004,A 0.000,B 0.000,C 90.000,E1 180.688} C_DIS
LIN {X 0.002,Y -141.229,Z 670.973,A 0.000,B 0.000,C 90.000,E1 175.122} C_DIS
LIN {X -0.039,Y -142.601,Z 670.957,A 0.000,B 0.000,C 90.000,E1 172.356} C_DIS
LIN {X 0.055,Y -144.909,Z 670.932,A 0.000,B 0.000,C 90.000,E1 167.701} C_DIS
LIN {X 0.007,Y -147.537,Z 670.911,A 0.000,B 0.000,C 90.000,E1 164.047} C_DIS
LIN {X -0.061,Y -150.136,Z 670.891,A 0.000,B 0.000,C 90.000,E1 160.423} C_DIS
LIN {X -0.050,Y -153.503,Z 670.871,A 0.000,B 0.000,C 90.000,E1 156.794} C_DIS
LIN {X 0.013,Y -157.867,Z 670.846,A 0.000,B 0.000,C 90.000,E1 152.281} C_DIS
LIN {X -0.032,Y -162.154,Z 670.826,A 0.000,B 0.000,C 90.000,E1 148.742} C_DIS
LIN {X 0.083,Y -166.359,Z 670.807,A 0.000,B 0.000,C 90.000,E1 145.182} C_DIS
LIN {X -0.048,Y -171.376,Z 670.787,A 0.000,B 0.000,C 90.000,E1 141.743} C_DIS
LIN {X -0.004,Y -176.286,Z 670.768,A 0.000,B 0.000,C 90.000,E1 138.286} C_DIS
LIN {X -0.004,Y -180.571,Z 670.754,A 0.000,B 0.000,C 90.000,E1 135.729} C_DIS
LIN {X -0.026,Y -185.973,Z 670.735,A 0.000,B 0.000,C 90.000,E1 132.366} C_DIS
LIN {X 0.059,Y -191.087,Z 670.720,A 0.000,B 0.000,C 90.000,E1 129.564} C_DIS
LIN {X 0.054,Y -289.130,Z 670.720,A 0.000,B 0.000,C 90.000,E1 129.564} C_DIS
LIN {X -0.020,Y -291.676,Z 670.720,A 0.000,B 0.000,C 90.000,E1 129.519} C_DIS
LIN {X -0.021,Y -295.880,Z 670.718,A 0.000,B 0.000,C 90.000,E1 129.277} C_DIS
LIN {X -0.022,Y -298.380,Z 670.717,A 0.000,B 0.000,C 90.000,E1 129.036} C_DIS
LIN {X 0.076,Y -302.146,Z 670.714,A 0.000,B 0.000,C 90.000,E1 128.463} C_DIS
LIN {X -0.164,Y -303.716,Z 670.712,A 0.000,B 0.000,C 90.000,E1 128.177} C_DIS
LIN {X 0.023,Y -304.951,Z 670.710,A 0.000,B 0.000,C 90.000,E1 127.810} C_DIS
LIN {X -0.069,Y -316.565,Z 670.688,A 0.000,B 0.000,C 90.000,E1 123.913} C_DIS
LIN {X 0.112,Y -326.642,Z 670.672,A 0.000,B 0.000,C 90.000,E1 121.003} C_DIS
LIN {X 0.093,Y -338.051,Z 670.657,A 0.000,B 0.000,C 90.000,E1 118.180} C_DIS
LIN {X 0.090,Y -350.888,Z 670.641,A 0.000,B 0.000,C 90.000,E1 115.412} C_DIS
LIN {X -0.070,Y -363.595,Z 670.628,A 0.000,B 0.000,C 90.000,E1 113.025} C_DIS
LIN {X -0.067,Y -377.616,Z 670.615,A 0.000,B 0.000,C 90.000,E1 110.663} C_DIS
LIN {X -0.118,Y -393.051,Z 670.602,A 0.000,B 0.000,C 90.000,E1 108.362} C_DIS
LIN {X 0.102,Y -410.013,Z 670.589,A 0.000,B 0.000,C 90.000,E1 106.079} C_DIS
